KUKA KRL program: MyProgram_304().src

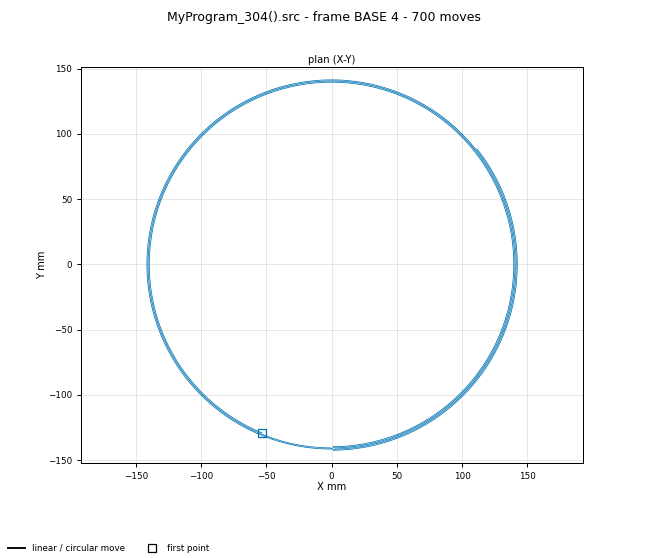
[picture p0: tool path of MyProgram_304().src in frame BASE 4, 700 of 700 moves have a stored position in this frame; points joined in program order, loops and branches not executed]
&ACCESS RVP
&REL 1
&PARAM TEMPLATE = C:\KRC\Roboter\Template\vorgabe
&PARAM EDITMASK = *
DEF MyProgram_304()
; ---- Setting reference (Base) ----
$BASE = BASE_DATA[4]

; --------------------------
; ---- Setting tool (TCP) ----
$TOOL = TOOL_DATA[3]
; --------------------------

$VEL.CP = VEL_APROX_PRINT
Startdeposition()
$VEL.CP = VEL_PRINT
LIN {X -53.4181,Y -129.0788,Z 180,A -108.7523,B 5.3109,C 0.3866,E1 5.2646,E2 201.3046} C_DIS
LIN {X -56.4505,Y -127.7825,Z 180,A -110.2013,B 5.3109,C 0.3863,E1 5.2608,E2 202.7664} C_DIS
LIN {X -60.7814,Y -125.7801,Z 180,A -112.5486,B 5.3109,C 0.3883,E1 5.2548,E2 205.165} C_DIS
LIN {X -64.8227,Y -123.7443,Z 180,A -113.8658,B 5.3114,C 0.3803,E1 5.2517,E2 206.4117} C_DIS
LIN {X -68.8662,Y -121.5434,Z 180,A -115.942,B 5.3114,C 0.3799,E1 5.2465,E2 208.5128} C_DIS
LIN {X -72.8889,Y -119.1739,Z 180,A -117.7837,B 5.3117,C 0.3765,E1 5.2422,E2 210.3448} C_DIS
LIN {X -75.6245,Y -117.4571,Z 180,A -119.198,B 5.3117,C 0.3756,E1 5.2388,E2 211.7709} C_DIS
LIN {X -78.8968,Y -115.2844,Z 180,A -121.1686,B 5.3117,C 0.3769,E1 5.2341,E2 213.7885} C_DIS
LIN {X -82.2269,Y -112.9324,Z 180,A -122.773,B 5.3119,C 0.3735,E1 5.2305,E2 215.384} C_DIS
LIN {X -85.2034,Y -110.7056,Z 180,A -124.0807,B 5.3122,C 0.3688,E1 5.2277,E2 216.6631} C_DIS
LIN {X -88.7338,Y -107.8966,Z 180,A -125.9867,B 5.3124,C 0.3662,E1 5.2235,E2 218.5762} C_DIS
LIN {X -92.192,Y -104.9572,Z 180,A -127.8448,B 5.3126,C 0.3629,E1 5.2196,E2 220.4335} C_DIS
LIN {X -95.4577,Y -101.9958,Z 180,A -129.699,B 5.3128,C 0.36,E1 5.2158,E2 222.2935} C_DIS
LIN {X -98.7586,Y -98.8033,Z 180,A -131.5928,B 5.313,C 0.3565,E1 5.212,E2 224.1882} C_DIS
LIN {X -101.9125,Y -95.5469,Z 180,A -133.5295,B 5.3132,C 0.3536,E1 5.2083,E2 226.1346} C_DIS
LIN {X -105.0138,Y -92.1271,Z 180,A -135.4558,B 5.3135,C 0.35,E1 5.2047,E2 228.0647} C_DIS
LIN {X -107.866,Y -88.7709,Z 180,A -137.2983,B 5.3137,C 0.3465,E1 5.2014,E2 229.9114} C_DIS
LIN {X -110.7145,Y -85.1918,Z 180,A -138.9304,B 5.3141,C 0.3401,E1 5.1986,E2 231.5111} C_DIS
LIN {X -112.3282,Y -83.0519,Z 180,A -140.3289,B 5.3141,C 0.3405,E1 5.1962,E2 232.9482} C_DIS
LIN {X -114.9154,Y -79.4344,Z 180,A -142.1992,B 5.3143,C 0.3368,E1 5.1932,E2 234.8238} C_DIS
LIN {X -116.9571,Y -76.3961,Z 180,A -143.832,B 5.3145,C 0.3345,E1 5.1907,E2 236.4731} C_DIS
LIN {X -119.7431,Y -71.9508,Z 180,A -145.7127,B 5.3149,C 0.3269,E1 5.188,E2 238.3177} C_DIS
LIN {X -122.8692,Y -66.4714,Z 180,A -148.6944,B 5.3151,C 0.3242,E1 5.1838,E2 241.3494} C_DIS
LIN {X -125.0963,Y -62.1747,Z 180,A -150.5037,B 5.3155,C 0.3177,E1 5.1816,E2 243.1351} C_DIS
LIN {X -126.6631,Y -58.9167,Z 180,A -152.1928,B 5.3156,C 0.3158,E1 5.1795,E2 244.8501} C_DIS
LIN {X -128.6518,Y -54.4406,Z 180,A -154.1647,B 5.3159,C 0.3103,E1 5.1773,E2 246.8163} C_DIS
LIN {X -129.8644,Y -51.4832,Z 180,A -155.7497,B 5.3159,C 0.3093,E1 5.1757,E2 248.4359} C_DIS
LIN {X -131.0841,Y -48.2916,Z 180,A -157.1548,B 5.3162,C 0.3056,E1 5.1743,E2 249.8406} C_DIS
LIN {X -132.1648,Y -45.2484,Z 180,A -158.3647,B 5.3165,C 0.3011,E1 5.1732,E2 251.035} C_DIS
LIN {X -133.3531,Y -41.62,Z 180,A -159.865,B 5.3167,C 0.2963,E1 5.1719,E2 252.5261} C_DIS
LIN {X -134.4327,Y -37.9823,Z 180,A -161.4301,B 5.317,C 0.2921,E1 5.1707,E2 254.0912} C_DIS
LIN {X -135.3964,Y -34.3875,Z 180,A -163.0135,B 5.3172,C 0.2885,E1 5.1696,E2 255.681} C_DIS
LIN {X -136.1324,Y -31.3482,Z 180,A -164.2721,B 5.3174,C 0.2847,E1 5.1688,E2 256.9357} C_DIS
LIN {X -136.8639,Y -27.9821,Z 180,A -165.5232,B 5.3176,C 0.2794,E1 5.1681,E2 258.1651} C_DIS
LIN {X -137.4255,Y -25.0834,Z 180,A -166.9887,B 5.3177,C 0.2783,E1 5.1673,E2 259.6626} C_DIS
LIN {X -138.0139,Y -21.6086,Z 180,A -168.4852,B 5.3179,C 0.2747,E1 5.1666,E2 261.1647} C_DIS
LIN {X -138.4562,Y -18.5685,Z 180,A -169.9672,B 5.3179,C 0.2731,E1 5.166,E2 262.6742} C_DIS
LIN {X -139.2639,Y -10.996,Z 180,A -173.1053,B 5.3184,C 0.2644,E1 5.1652,E2 265.812} C_DIS
LIN {X -139.4901,Y -7.5904,Z 180,A -174.8697,B 5.3184,C 0.2636,E1 5.1649,E2 267.6217} C_DIS
LIN {X -139.6482,Y -3.635,Z 180,A -175.7772,B 5.319,C 0.2527,E1 5.1649,E2 268.4367} C_DIS
LIN {X -139.6884,Y 1.5471,Z 180,A -178.478,B 5.319,C 0.2517,E1 5.1649,E2 271.2095} C_DIS
LIN {X -139.3259,Y 10.151,Z 180,A 178.1814,B 5.3196,C 0.24,E1 5.1653,E2 274.523} C_DIS
LIN {X -138.7226,Y 16.4559,Z 180,A 175.3926,B 5.3198,C 0.2343,E1 5.166,E2 277.3342} C_DIS
LIN {X -138.2382,Y 20.1258,Z 180,A 173.8815,B 5.32,C 0.2299,E1 5.1666,E2 278.8431} C_DIS
LIN {X -137.7937,Y 22.9699,Z 180,A 172.4203,B 5.32,C 0.229,E1 5.1673,E2 280.3389} C_DIS
LIN {X -136.6551,Y 28.9886,Z 180,A 170.1284,B 5.3204,C 0.2201,E1 5.1685,E2 282.6008} C_DIS
LIN {X -135.9071,Y 32.3133,Z 180,A 168.5489,B 5.3205,C 0.2178,E1 5.1695,E2 284.2022} C_DIS
LIN {X -135.0439,Y 35.7475,Z 180,A 167.0737,B 5.3207,C 0.214,E1 5.1705,E2 285.679} C_DIS
LIN {X -134.221,Y 38.7258,Z 180,A 165.7742,B 5.3207,C 0.2108,E1 5.1715,E2 286.9816} C_DIS
LIN {X -133.127,Y 42.3307,Z 180,A 164.1851,B 5.3209,C 0.207,E1 5.1729,E2 288.5749} C_DIS
LIN {X -131.7274,Y 46.5099,Z 180,A 162.2401,B 5.3211,C 0.2033,E1 5.1746,E2 290.5357} C_DIS
LIN {X -130.6009,Y 49.5825,Z 180,A 160.8237,B 5.3211,C 0.2004,E1 5.1761,E2 291.9603} C_DIS
LIN {X -128.5842,Y 54.6025,Z 180,A 158.5967,B 5.3214,C 0.1946,E1 5.1784,E2 294.1864} C_DIS
LIN {X -126.939,Y 58.3201,Z 180,A 157.2078,B 5.3217,C 0.1878,E1 5.18,E2 295.5387} C_DIS
LIN {X -125.701,Y 60.9469,Z 180,A 155.4772,B 5.3216,C 0.1895,E1 5.1821,E2 297.3362} C_DIS
LIN {X -124.2165,Y 63.9159,Z 180,A 154.1121,B 5.3217,C 0.1861,E1 5.1839,E2 298.7005} C_DIS
LIN {X -122.6686,Y 66.8402,Z 180,A 152.908,B 5.3219,C 0.1814,E1 5.1854,E2 299.8843} C_DIS
LIN {X -120.3453,Y 70.9383,Z 180,A 150.9383,B 5.322,C 0.1769,E1 5.1882,E2 301.8571} C_DIS
LIN {X -117.9862,Y 74.7965,Z 180,A 149.0261,B 5.3222,C 0.173,E1 5.191,E2 303.7748} C_DIS
LIN {X -115.4538,Y 78.6496,Z 180,A 147.077,B 5.3222,C 0.169,E1 5.1941,E2 305.7295} C_DIS
LIN {X -112.8106,Y 82.3959,Z 180,A 145.3761,B 5.3225,C 0.163,E1 5.1968,E2 307.4063} C_DIS
LIN {X -110.0024,Y 86.1086,Z 180,A 143.1989,B 5.3225,C 0.1612,E1 5.2005,E2 309.6154} C_DIS
LIN {X -107.1393,Y 89.6459,Z 180,A 141.4016,B 5.3227,C 0.1565,E1 5.2037,E2 311.4025} C_DIS
LIN {X -103.7343,Y 93.5651,Z 180,A 138.6523,B 5.3227,C 0.1577,E1 5.209,E2 314.227} C_DIS
LIN {X -100.4211,Y 97.1123,Z 180,A 137.1074,B 5.3229,C 0.1495,E1 5.2118,E2 315.715} C_DIS
LIN {X -97.8974,Y 99.6558,Z 180,A 135.0674,B 5.3228,C 0.1519,E1 5.216,E2 317.8245} C_DIS
LIN {X -94.1292,Y 103.223,Z 180,A 132.9812,B 5.3229,C 0.1475,E1 5.2203,E2 319.9038} C_DIS
LIN {X -90.597,Y 106.3362,Z 180,A 131.4762,B 5.3231,C 0.1399,E1 5.2234,E2 321.3544} C_DIS
LIN {X -87.0706,Y 109.2423,Z 180,A 129.612,B 5.3232,C 0.1364,E1 5.2274,E2 323.2158} C_DIS
LIN {X -84.1015,Y 111.5443,Z 180,A 127.5305,B 5.3232,C 0.1391,E1 5.2322,E2 325.3631} C_DIS
LIN {X -80.1977,Y 114.3838,Z 180,A 125.9877,B 5.3233,C 0.1316,E1 5.2356,E2 326.8502} C_DIS
LIN {X -76.4605,Y 116.9152,Z 180,A 124.1034,B 5.3234,C 0.129,E1 5.24,E2 328.7372} C_DIS
LIN {X -72.6594,Y 119.3147,Z 180,A 122.36,B 5.3234,C 0.1253,E1 5.2441,E2 330.4667} C_DIS
LIN {X -69.4823,Y 121.1919,Z 180,A 120.6836,B 5.3235,C 0.1248,E1 5.2482,E2 332.1622} C_DIS
LIN {X -65.5195,Y 123.3784,Z 180,A 118.8849,B 5.3235,C 0.1218,E1 5.2526,E2 333.9523} C_DIS
LIN {X -62.1192,Y 125.1237,Z 180,A 117.2852,B 5.3236,C 0.1201,E1 5.2566,E2 335.5548} C_DIS
LIN {X -57.8735,Y 127.1455,Z 180,A 115.2756,B 5.3236,C 0.1187,E1 5.2617,E2 337.5732} C_DIS
LIN {X -51.9459,Y 129.6779,Z 180,A 112.3818,B 5.3236,C 0.1185,E1 5.2692,E2 340.496} C_DIS
LIN {X -48.6279,Y 130.9585,Z 180,A 111.18,B 5.3237,C 0.1144,E1 5.2723,E2 341.665} C_DIS
LIN {X -44.4366,Y 132.4392,Z 180,A 109.372,B 5.3237,C 0.1126,E1 5.277,E2 343.4699} C_DIS
LIN {X -41.3217,Y 133.4443,Z 180,A 108.0284,B 5.3237,C 0.1115,E1 5.2806,E2 344.8128} C_DIS
LIN {X -38.2459,Y 134.359,Z 180,A 106.3124,B 5.3237,C 0.1148,E1 5.2854,E2 346.5775} C_DIS
LIN {X -34.5071,Y 135.366,Z 180,A 105.1143,B 5.3238,C 0.1096,E1 5.2885,E2 347.7263} C_DIS
LIN {X -31.3524,Y 136.1315,Z 180,A 103.7636,B 5.3238,C 0.109,E1 5.2921,E2 349.0787} C_DIS
LIN {X -28.0893,Y 136.8421,Z 180,A 102.2931,B 5.3238,C 0.1093,E1 5.2962,E2 350.5609} C_DIS
LIN {X -19.2145,Y 138.3685,Z 180,A 98.5818,B 5.3238,C 0.108,E1 5.3064,E2 354.2724} C_DIS
LIN {X -15.0864,Y 138.8782,Z 180,A 96.9214,B 5.3238,C 0.107,E1 5.311,E2 355.9262} C_DIS
LIN {X -9.6565,Y 139.362,Z 180,A 94.5696,B 5.3238,C 0.1079,E1 5.3176,E2 358.2914} C_DIS
LIN {X -5.0259,Y 139.6055,Z 180,A 92.8427,B 5.3239,C 0.1057,E1 5.3224,E2 359.9957} C_DIS
LIN {X -1.2399,Y 139.6906,Z 180,A 91.2064,B 5.3239,C 0.1067,E1 5.327,E2 361.6416} C_DIS
LIN {X 3.0957,Y 139.6631,Z 180,A 89.4454,B 5.3239,C 0.1067,E1 5.3319,E2 363.3998} C_DIS
LIN {X 6.8555,Y 139.527,Z 180,A 87.9816,B 5.3239,C 0.1059,E1 5.3359,E2 364.853} C_DIS
LIN {X 10.1316,Y 139.3273,Z 180,A 86.6321,B 5.3239,C 0.1063,E1 5.3397,E2 366.2023} C_DIS
LIN {X 13.9379,Y 138.9994,Z 180,A 84.9893,B 5.3239,C 0.1077,E1 5.3443,E2 367.854} C_DIS
LIN {X 17.3009,Y 138.6217,Z 180,A 83.4925,B 5.3239,C 0.1095,E1 5.3485,E2 369.3639} C_DIS
LIN {X 23.4985,Y 137.7055,Z 180,A 81.0194,B 5.3239,C 0.1095,E1 5.3553,E2 371.8242} C_DIS
LIN {X 27.313,Y 137,Z 180,A 79.39,B 5.3239,C 0.111,E1 5.3597,E2 373.4579} C_DIS
LIN {X 31.8403,Y 136.0189,Z 180,A 77.378,B 5.3238,C 0.1136,E1 5.3653,E2 375.4832} C_DIS
LIN {X 35.117,Y 135.2112,Z 180,A 76.2143,B 5.3238,C 0.1119,E1 5.3683,E2 376.6193} C_DIS
LIN {X 38.9715,Y 134.1491,Z 180,A 74.6646,B 5.3238,C 0.1121,E1 5.3725,E2 378.1573} C_DIS
LIN {X 41.8856,Y 133.2692,Z 180,A 73.3079,B 5.3238,C 0.1146,E1 5.3761,E2 379.5274} C_DIS
LIN {X 46.6217,Y 131.6879,Z 180,A 71.2783,B 5.3237,C 0.1163,E1 5.3815,E2 381.5543} C_DIS
LIN {X 50.0811,Y 130.4103,Z 180,A 69.8417,B 5.3237,C 0.1169,E1 5.3852,E2 382.9812} C_DIS
LIN {X 53.5107,Y 129.0401,Z 180,A 68.3385,B 5.3237,C 0.1185,E1 5.3891,E2 384.4828} C_DIS
LIN {X 56.8677,Y 127.5959,Z 180,A 67.0037,B 5.3237,C 0.1181,E1 5.3924,E2 385.7969} C_DIS
LIN {X 62.2697,Y 125.0495,Z 180,A 64.5146,B 5.3236,C 0.1217,E1 5.3987,E2 388.2908} C_DIS
LIN {X 66.0051,Y 123.12,Z 180,A 62.6956,B 5.3235,C 0.1253,E1 5.4033,E2 390.1216} C_DIS
LIN {X 70.0877,Y 120.8425,Z 180,A 60.8254,B 5.3235,C 0.1274,E1 5.4078,E2 391.9859} C_DIS
LIN {X 74.0028,Y 118.4856,Z 180,A 58.9975,B 5.3234,C 0.1296,E1 5.4121,E2 393.808} C_DIS
LIN {X 77.581,Y 116.1739,Z 180,A 56.9544,B 5.3232,C 0.1364,E1 5.417,E2 395.8882} C_DIS
LIN {X 80.7286,Y 114.0094,Z 180,A 55.6359,B 5.3232,C 0.1356,E1 5.4199,E2 397.1758} C_DIS
LIN {X 84.5976,Y 111.169,Z 180,A 53.724,B 5.3232,C 0.1382,E1 5.4242,E2 399.0807} C_DIS
LIN {X 88.2382,Y 108.3016,Z 180,A 51.827,B 5.3231,C 0.1416,E1 5.4283,E2 400.9775} C_DIS
LIN {X 92.0568,Y 105.0752,Z 180,A 49.9356,B 5.3231,C 0.1433,E1 5.4323,E2 402.8493} C_DIS
LIN {X 94.5696,Y 102.8191,Z 180,A 47.9785,B 5.3227,C 0.1539,E1 5.4365,E2 404.8782} C_DIS
LIN {X 98.3552,Y 99.2041,Z 180,A 46.3995,B 5.3228,C 0.1503,E1 5.4395,E2 406.3866} C_DIS
LIN {X 101.5988,Y 95.8794,Z 180,A 44.5516,B 5.3228,C 0.1534,E1 5.443,E2 408.2278} C_DIS
LIN {X 104.6892,Y 92.4951,Z 180,A 42.7152,B 5.3227,C 0.1568,E1 5.4465,E2 410.0592} C_DIS
LIN {X 107.1038,Y 89.6882,Z 180,A 40.9069,B 5.3224,C 0.1642,E1 5.4498,E2 411.9043} C_DIS
LIN {X 109.6071,Y 86.6119,Z 180,A 39.586,B 5.3224,C 0.1635,E1 5.452,E2 413.1873} C_DIS
LIN {X 112.3135,Y 83.0726,Z 180,A 37.8081,B 5.3224,C 0.167,E1 5.455,E2 414.9596} C_DIS
LIN {X 114.8587,Y 79.5158,Z 180,A 36.1736,B 5.3223,C 0.1689,E1 5.4576,E2 416.5745} C_DIS
LIN {X 116.9308,Y 76.4366,Z 180,A 34.5411,B 5.3221,C 0.1741,E1 5.4601,E2 418.2216} C_DIS
LIN {X 118.9321,Y 73.2831,Z 180,A 32.8039,B 5.3219,C 0.1808,E1 5.4627,E2 419.9854} C_DIS
LIN {X 120.8792,Y 70.0239,Z 180,A 31.4886,B 5.3219,C 0.1811,E1 5.4645,E2 421.2707} C_DIS
LIN {X 123.2434,Y 65.7753,Z 180,A 29.5782,B 5.3218,C 0.1849,E1 5.4671,E2 423.1714} C_DIS
LIN {X 125.0282,Y 62.3128,Z 180,A 28.2508,B 5.3218,C 0.1849,E1 5.4687,E2 424.4651} C_DIS
LIN {X 126.6486,Y 58.948,Z 180,A 26.6413,B 5.3216,C 0.1901,E1 5.4706,E2 426.0853} C_DIS
LIN {X 128.0692,Y 55.7949,Z 180,A 25.4362,B 5.3216,C 0.1906,E1 5.472,E2 427.2639} C_DIS
LIN {X 130.2404,Y 50.5183,Z 180,A 23.0133,B 5.3213,C 0.198,E1 5.4746,E2 429.6986} C_DIS
LIN {X 131.3973,Y 47.4278,Z 180,A 21.7673,B 5.3213,C 0.2,E1 5.4757,E2 430.9317} C_DIS
LIN {X 132.4219,Y 44.4886,Z 180,A 20.423,B 5.321,C 0.2045,E1 5.477,E2 432.2854} C_DIS
LIN {X 133.5287,Y 41.046,Z 180,A 18.9479,B 5.3209,C 0.2084,E1 5.4782,E2 433.7603} C_DIS
LIN {X 134.5026,Y 37.7326,Z 180,A 17.6107,B 5.3208,C 0.2111,E1 5.4792,E2 435.0882} C_DIS
LIN {X 135.3467,Y 34.5835,Z 180,A 16.2761,B 5.3206,C 0.2147,E1 5.4802,E2 436.4233} C_DIS
LIN {X 136.0439,Y 31.7359,Z 180,A 15.1574,B 5.3206,C 0.2168,E1 5.4809,E2 437.532} C_DIS
LIN {X 136.9679,Y 27.471,Z 180,A 13.2708,B 5.3203,C 0.2232,E1 5.482,E2 439.4322} C_DIS
LIN {X 137.6674,Y 23.727,Z 180,A 11.1723,B 5.3198,C 0.2356,E1 5.483,E2 441.6003} C_DIS
LIN {X 138.492,Y 18.2952,Z 180,A 9.5426,B 5.3198,C 0.2326,E1 5.4836,E2 443.1519} C_DIS
LIN {X 139.0361,Y 13.5554,Z 180,A 7.728,B 5.3198,C 0.236,E1 5.4841,E2 444.9496} C_DIS
LIN {X 139.3314,Y 10.0758,Z 180,A 6.3138,B 5.3196,C 0.2398,E1 5.4844,E2 446.3625} C_DIS
LIN {X 139.5729,Y 5.8598,Z 180,A 4.6384,B 5.3194,C 0.2439,E1 5.4847,E2 448.0319} C_DIS
LIN {X 139.6755,Y 2.3565,Z 180,A 3.267,B 5.3192,C 0.247,E1 5.4847,E2 449.3957} C_DIS
LIN {X 139.6814,Y -1.9962,Z 180,A 1.495,B 5.319,C 0.2519,E1 5.4847,E2 451.1675} C_DIS
LIN {X 139.5624,Y -6.1305,Z 180,A -0.2183,B 5.3188,C 0.257,E1 5.4846,E2 452.8842} C_DIS
LIN {X 139.3144,Y -10.3093,Z 180,A -1.8235,B 5.3186,C 0.2602,E1 5.4843,E2 454.4764} C_DIS
LIN {X 138.932,Y -14.5868,Z 180,A -3.5823,B 5.3184,C 0.2651,E1 5.4838,E2 456.2362} C_DIS
LIN {X 138.4803,Y -18.3843,Z 180,A -5.0577,B 5.3182,C 0.2682,E1 5.4833,E2 457.7008} C_DIS
LIN {X 137.8848,Y -22.4237,Z 180,A -7.1758,B 5.3176,C 0.2796,E1 5.4823,E2 459.8776} C_DIS
LIN {X 137.0513,Y -27.0612,Z 180,A -8.6435,B 5.3177,C 0.278,E1 5.4816,E2 461.287} C_DIS
LIN {X 136.2801,Y -30.7018,Z 180,A -10.0627,B 5.3176,C 0.2807,E1 5.4807,E2 462.6935} C_DIS
LIN {X 134.9928,Y -35.9392,Z 180,A -12.0724,B 5.3174,C 0.2837,E1 5.4794,E2 464.6787} C_DIS
LIN {X 133.1515,Y -42.2542,Z 180,A -14.8183,B 5.317,C 0.2919,E1 5.4772,E2 467.4332} C_DIS
LIN {X 132.0483,Y -45.5842,Z 180,A -16.2158,B 5.3168,C 0.2952,E1 5.476,E2 468.8266} C_DIS
LIN {X 130.9944,Y -48.5319,Z 180,A -17.5271,B 5.3166,C 0.2991,E1 5.4747,E2 470.1426} C_DIS
LIN {X 129.6758,Y -51.951,Z 180,A -18.8882,B 5.3165,C 0.301,E1 5.4733,E2 471.4864} C_DIS
LIN {X 128.3506,Y -55.144,Z 180,A -20.2885,B 5.3163,C 0.3045,E1 5.4718,E2 472.8857} C_DIS
LIN {X 126.9225,Y -58.3557,Z 180,A -21.7176,B 5.3161,C 0.3081,E1 5.4702,E2 474.3145} C_DIS
LIN {X 125.5516,Y -61.2518,Z 180,A -23.069,B 5.3158,C 0.312,E1 5.4685,E2 475.6719} C_DIS
LIN {X 123.7294,Y -64.8509,Z 180,A -24.6078,B 5.3157,C 0.3146,E1 5.4666,E2 477.197} C_DIS
LIN {X 121.6076,Y -68.7525,Z 180,A -26.4799,B 5.3154,C 0.3199,E1 5.464,E2 479.0774} C_DIS
LIN {X 119.4654,Y -72.4101,Z 180,A -28.5865,B 5.3148,C 0.3297,E1 5.4609,E2 481.2336} C_DIS
LIN {X 117.0766,Y -76.212,Z 180,A -29.9613,B 5.3149,C 0.3273,E1 5.459,E2 482.5491} C_DIS
LIN {X 114.5875,Y -79.9056,Z 180,A -31.6688,B 5.3148,C 0.3299,E1 5.4563,E2 484.2426} C_DIS
LIN {X 112.2867,Y -83.1086,Z 180,A -33.9984,B 5.3139,C 0.3442,E1 5.4523,E2 486.6666} C_DIS
LIN {X 108.717,Y -87.7256,Z 180,A -35.6708,B 5.3142,C 0.3391,E1 5.4495,E2 488.2471} C_DIS
LIN {X 105.9713,Y -91.0236,Z 180,A -37.3819,B 5.314,C 0.3423,E1 5.4464,E2 489.9533} C_DIS
LIN {X 104.0082,Y -93.2603,Z 180,A -38.6493,B 5.3138,C 0.3457,E1 5.4441,E2 491.2279} C_DIS
LIN {X 101.3904,Y -96.1003,Z 180,A -40.1605,B 5.3136,C 0.348,E1 5.4412,E2 492.7309} C_DIS
LIN {X 98.3275,Y -99.2317,Z 180,A -41.8803,B 5.3134,C 0.3507,E1 5.4378,E2 494.4421} C_DIS
LIN {X 95.3265,Y -102.1179,Z 180,A -43.6035,B 5.3132,C 0.3544,E1 5.4343,E2 496.1689} C_DIS
LIN {X 92.019,Y -105.1082,Z 180,A -45.2382,B 5.3132,C 0.3552,E1 5.431,E2 497.7796} C_DIS
LIN {X 89.2239,Y -107.4909,Z 180,A -46.8661,B 5.3128,C 0.3598,E1 5.4275,E2 499.4248} C_DIS
LIN {X 85.8046,Y -110.2399,Z 180,A -48.3533,B 5.3128,C 0.3587,E1 5.4243,E2 500.8722} C_DIS
LIN {X 83.6515,Y -111.8824,Z 180,A -49.6148,B 5.3126,C 0.3629,E1 5.4214,E2 502.1547} C_DIS
LIN {X 79.6876,Y -114.7392,Z 180,A -51.7708,B 5.3122,C 0.3685,E1 5.4165,E2 504.3323} C_DIS
LIN {X 75.6663,Y -117.4307,Z 180,A -53.9476,B 5.3118,C 0.3745,E1 5.4113,E2 506.536} C_DIS
LIN {X 72.4638,Y -119.4329,Z 180,A -54.965,B 5.3122,C 0.3695,E1 5.4091,E2 507.4846} C_DIS
LIN {X 67.1571,Y -122.4957,Z 180,A -57.6945,B 5.3117,C 0.3763,E1 5.4024,E2 510.2447} C_DIS
LIN {X 63.5525,Y -124.4015,Z 180,A -59.2118,B 5.3117,C 0.3765,E1 5.3987,E2 511.7428} C_DIS
LIN {X 60.3887,Y -125.9677,Z 180,A -60.674,B 5.3115,C 0.3787,E1 5.395,E2 513.208} C_DIS
LIN {X 57.1271,Y -127.4799,Z 180,A -61.9984,B 5.3115,C 0.3786,E1 5.3917,E2 514.5136} C_DIS
LIN {X 54.1683,Y -128.7655,Z 180,A -63.3875,B 5.3113,C 0.3811,E1 5.3881,E2 515.9124} C_DIS
LIN {X 50.9744,Y -130.063,Z 180,A -64.8485,B 5.3112,C 0.3834,E1 5.3843,E2 517.3806} C_DIS
LIN {X 47.7036,Y -131.2979,Z 180,A -66.2567,B 5.3111,C 0.3846,E1 5.3806,E2 518.7865} C_DIS
LIN {X 44.2513,Y -132.5009,Z 180,A -67.7178,B 5.3111,C 0.3856,E1 5.3767,E2 520.2435} C_DIS
LIN {X 41.1267,Y -133.504,Z 180,A -68.8889,B 5.3111,C 0.3846,E1 5.3737,E2 521.3923} C_DIS
LIN {X 37.023,Y -134.701,Z 180,A -70.8902,B 5.3107,C 0.3895,E1 5.3682,E2 523.4278} C_DIS
LIN {X 30.5957,Y -136.3043,Z 180,A -73.5088,B 5.3107,C 0.3904,E1 5.3611,E2 526.0351} C_DIS
LIN {X 23.7366,Y -137.6657,Z 180,A -76.8393,B 5.3101,C 0.3982,E1 5.3518,E2 529.4284} C_DIS
LIN {X 19.4208,Y -138.339,Z 180,A -78.1847,B 5.3104,C 0.3934,E1 5.3483,E2 530.7159} C_DIS
LIN {X 15.4627,Y -138.8377,Z 180,A -79.8042,B 5.3104,C 0.394,E1 5.3438,E2 532.3341} C_DIS
LIN {X 11.8735,Y -139.1897,Z 180,A -81.2565,B 5.3104,C 0.3942,E1 5.3397,E2 533.7836} C_DIS
LIN {X 7.819,Y -139.4783,Z 180,A -82.9889,B 5.3103,C 0.3955,E1 5.3349,E2 535.5256} C_DIS
LIN {X 3.6418,Y -139.648,Z 180,A -84.6179,B 5.3103,C 0.3949,E1 5.3304,E2 537.1441} C_DIS
LIN {X 0.988,Y -139.6903,Z 180,A -85.5323,B 5.3105,C 0.3929,E1 5.3279,E2 538.0358} C_DIS
Enddeposition()
LIN {X 0.988,Y -139.6903,Z 180,A -85.5323,B 5.3105,C 0.3929,E1 5.3279,E2 538.0358} C_DIS
Startdeposition()
$VEL.CP = VEL_PRINT
LIN {X 1.6591,Y -140.5898,Z 180,A -84.529,B 5.0673,C 0.3825,E1 5.0873,E2 537.0364} C_DIS
LIN {X 5.6051,Y -140.4862,Z 180,A -83.0223,B 5.0673,C 0.3834,E1 5.0914,E2 535.5427} C_DIS
LIN {X 9.7167,Y -140.2627,Z 180,A -81.2945,B 5.0673,C 0.3822,E1 5.0963,E2 533.8074} C_DIS
LIN {X 13.6344,Y -139.9353,Z 180,A -79.7585,B 5.0673,C 0.3824,E1 5.1005,E2 532.2794} C_DIS
LIN {X 17.757,Y -139.4729,Z 180,A -77.6117,B 5.0678,C 0.3759,E1 5.1067,E2 530.0698} C_DIS
LIN {X 22.0608,Y -138.8573,Z 180,A -76.277,B 5.0675,C 0.3804,E1 5.1102,E2 528.7934} C_DIS
LIN {X 26.0361,Y -138.1665,Z 180,A -74.5889,B 5.0675,C 0.3788,E1 5.1148,E2 527.0984} C_DIS
LIN {X 29.9679,Y -137.3671,Z 180,A -72.4377,B 5.0682,C 0.3711,E1 5.1209,E2 524.876} C_DIS
LIN {X 35.0666,Y -136.1553,Z 180,A -70.9688,B 5.0677,C 0.3779,E1 5.1247,E2 523.4964} C_DIS
LIN {X 38.4418,Y -135.2415,Z 180,A -69.2728,B 5.068,C 0.3732,E1 5.1293,E2 521.7628} C_DIS
LIN {X 43.0773,Y -133.8361,Z 180,A -67.5594,B 5.0679,C 0.3746,E1 5.1338,E2 520.0833} C_DIS
LIN {X 46.4412,Y -132.7066,Z 180,A -66.135,B 5.0679,C 0.3734,E1 5.1375,E2 518.6608} C_DIS
LIN {X 49.962,Y -131.4227,Z 180,A -64.6541,B 5.0681,C 0.3723,E1 5.1414,E2 517.1851} C_DIS
LIN {X 52.7883,Y -130.3115,Z 180,A -63.3956,B 5.0681,C 0.3706,E1 5.1447,E2 515.9228} C_DIS
LIN {X 56.5308,Y -128.7344,Z 180,A -61.7768,B 5.0683,C 0.369,E1 5.1488,E2 514.3078} C_DIS
LIN {X 59.2753,Y -127.4918,Z 180,A -60.5485,B 5.0684,C 0.3674,E1 5.1519,E2 513.0785} C_DIS
LIN {X 62.7104,Y -125.8386,Z 180,A -59.0283,B 5.0685,C 0.3658,E1 5.1558,E2 511.5616} C_DIS
LIN {X 65.3966,Y -124.4624,Z 180,A -57.847,B 5.0686,C 0.3647,E1 5.1587,E2 510.3859} C_DIS
LIN {X 69.9432,Y -121.9681,Z 180,A -55.4729,B 5.0691,C 0.358,E1 5.1645,E2 507.975} C_DIS
LIN {X 75.4813,Y -118.6209,Z 180,A -53.3038,B 5.0689,C 0.3602,E1 5.1696,E2 505.867} C_DIS
LIN {X 78.1143,Y -116.9032,Z 180,A -51.3428,B 5.0697,C 0.3487,E1 5.1743,E2 503.813} C_DIS
LIN {X 82.015,Y -114.2005,Z 180,A -49.8294,B 5.0696,C 0.3512,E1 5.1777,E2 502.3551} C_DIS
LIN {X 85.9243,Y -111.2891,Z 180,A -47.9606,B 5.0697,C 0.3492,E1 5.1818,E2 500.5005} C_DIS
LIN {X 89.0765,Y -108.7823,Z 180,A -46.359,B 5.0699,C 0.3467,E1 5.1852,E2 498.9029} C_DIS
LIN {X 92.8247,Y -105.6026,Z 180,A -44.3228,B 5.0702,C 0.3424,E1 5.1896,E2 496.8605} C_DIS
LIN {X 96.2359,Y -102.5035,Z 180,A -42.5076,B 5.0704,C 0.3395,E1 5.1933,E2 495.0522} C_DIS
LIN {X 99.4726,Y -99.3657,Z 180,A -40.6808,B 5.0706,C 0.3358,E1 5.1969,E2 493.2252} C_DIS
LIN {X 103.7158,Y -94.9276,Z 180,A -38.2282,B 5.0709,C 0.3312,E1 5.2016,E2 490.7772} C_DIS
LIN {X 106.7536,Y -91.4985,Z 180,A -36.4138,B 5.0711,C 0.3278,E1 5.2049,E2 488.9681} C_DIS
LIN {X 109.6839,Y -87.9646,Z 180,A -34.3051,B 5.0716,C 0.3201,E1 5.2087,E2 486.8258} C_DIS
LIN {X 112.0988,Y -84.8651,Z 180,A -32.9868,B 5.0716,C 0.3205,E1 5.2108,E2 485.5441} C_DIS
LIN {X 117.0782,Y -77.8522,Z 180,A -29.8517,B 5.0718,C 0.3175,E1 5.2158,E2 482.4557} C_DIS
LIN {X 120.6294,Y -72.2276,Z 180,A -27.0992,B 5.0722,C 0.3103,E1 5.2199,E2 479.6954} C_DIS
LIN {X 122.5106,Y -68.9881,Z 180,A -25.4793,B 5.0725,C 0.3051,E1 5.2221,E2 478.0617} C_DIS
LIN {X 124.6716,Y -64.9983,Z 180,A -23.7439,B 5.0727,C 0.302,E1 5.2244,E2 476.3399} C_DIS
LIN {X 126.2382,Y -61.9003,Z 180,A -22.3939,B 5.0729,C 0.2993,E1 5.2261,E2 474.9972} C_DIS
LIN {X 127.7298,Y -58.7605,Z 180,A -20.9869,B 5.0731,C 0.2958,E1 5.2277,E2 473.5902} C_DIS
LIN {X 129.1559,Y -55.556,Z 180,A -19.5724,B 5.0733,C 0.2922,E1 5.2293,E2 472.1764} C_DIS
LIN {X 130.7266,Y -51.7586,Z 180,A -17.8413,B 5.0736,C 0.2869,E1 5.2311,E2 470.4364} C_DIS
LIN {X 132.1842,Y -47.9067,Z 180,A -16.3399,B 5.0737,C 0.285,E1 5.2326,E2 468.9571} C_DIS
LIN {X 133.353,Y -44.5496,Z 180,A -14.9465,B 5.0739,C 0.2819,E1 5.2338,E2 467.5698} C_DIS
LIN {X 134.8138,Y -39.9137,Z 180,A -12.6642,B 5.0744,C 0.272,E1 5.2357,E2 465.2457} C_DIS
LIN {X 135.8091,Y -36.3812,Z 180,A -10.9466,B 5.0748,C 0.2645,E1 5.2369,E2 463.4971} C_DIS
LIN {X 137.0637,Y -31.3248,Z 180,A -9.5821,B 5.0745,C 0.2699,E1 5.2378,E2 462.2319} C_DIS
LIN {X 138.6594,Y -23.2659,Z 180,A -6.4873,B 5.0748,C 0.2643,E1 5.2394,E2 459.1681} C_DIS
LIN {X 139.262,Y -19.3423,Z 180,A -4.6833,B 5.0752,C 0.257,E1 5.2401,E2 457.3383} C_DIS
LIN {X 139.7411,Y -15.5049,Z 180,A -3.0438,B 5.0755,C 0.2516,E1 5.2407,E2 455.6891} C_DIS
LIN {X 140.1172,Y -11.6184,Z 180,A -1.5954,B 5.0755,C 0.2492,E1 5.241,E2 454.2584} C_DIS
LIN {X 140.3475,Y -8.3912,Z 180,A -0.2573,B 5.0758,C 0.2451,E1 5.2413,E2 452.9167} C_DIS
LIN {X 140.5382,Y -4.1036,Z 180,A 1.4403,B 5.076,C 0.2409,E1 5.2415,E2 451.2244} C_DIS
LIN {X 140.6015,Y -0.0685,Z 180,A 3.1089,B 5.0762,C 0.2359,E1 5.2415,E2 449.5516} C_DIS
LIN {X 140.5487,Y 3.7249,Z 180,A 4.529,B 5.0763,C 0.2333,E1 5.2415,E2 448.1469} C_DIS
LIN {X 140.3989,Y 7.4915,Z 180,A 5.9684,B 5.0765,C 0.2304,E1 5.2412,E2 446.7191} C_DIS
LIN {X 140.1559,Y 11.1598,Z 180,A 7.5796,B 5.0767,C 0.2245,E1 5.2409,E2 445.0919} C_DIS
LIN {X 139.7915,Y 15.0361,Z 180,A 9.8258,B 5.0773,C 0.2102,E1 5.2402,E2 442.7573} C_DIS
LIN {X 138.9564,Y 21.4209,Z 180,A 11.3602,B 5.077,C 0.219,E1 5.2396,E2 441.365} C_DIS
LIN {X 138.4135,Y 24.6866,Z 180,A 12.8764,B 5.0772,C 0.2127,E1 5.2389,E2 439.8261} C_DIS
LIN {X 137.6453,Y 28.6688,Z 180,A 14.4278,B 5.0774,C 0.2096,E1 5.2381,E2 438.287} C_DIS
LIN {X 137.0158,Y 31.5344,Z 180,A 15.7867,B 5.0776,C 0.2039,E1 5.2372,E2 436.9059} C_DIS
LIN {X 135.71,Y 36.753,Z 180,A 17.7502,B 5.0777,C 0.2012,E1 5.2359,E2 434.971} C_DIS
LIN {X 134.8797,Y 39.6886,Z 180,A 19.0202,B 5.0779,C 0.1974,E1 5.2349,E2 433.6967} C_DIS
LIN {X 133.8341,Y 43.0836,Z 180,A 20.4031,B 5.0779,C 0.1944,E1 5.2337,E2 432.3215} C_DIS
LIN {X 132.5866,Y 46.7873,Z 180,A 21.946,B 5.0781,C 0.1909,E1 5.2323,E2 430.7843} C_DIS
LIN {X 130.1483,Y 53.1933,Z 180,A 24.6707,B 5.0783,C 0.1845,E1 5.2296,E2 428.067} C_DIS
LIN {X 128.9303,Y 56.0778,Z 180,A 25.9136,B 5.0784,C 0.1816,E1 5.2282,E2 426.8278} C_DIS
LIN {X 127.4724,Y 59.3172,Z 180,A 27.3389,B 5.0786,C 0.1782,E1 5.2265,E2 425.4047} C_DIS
LIN {X 125.9366,Y 62.5117,Z 180,A 28.7637,B 5.0786,C 0.1748,E1 5.2248,E2 423.9818} C_DIS
LIN {X 124.0201,Y 66.2369,Z 180,A 30.5188,B 5.0789,C 0.1698,E1 5.2225,E2 422.2197} C_DIS
LIN {X 120.7546,Y 72.0176,Z 180,A 32.7789,B 5.0789,C 0.1695,E1 5.2195,E2 420.0162} C_DIS
LIN {X 118.0141,Y 76.4257,Z 180,A 35.2036,B 5.0792,C 0.16,E1 5.2158,E2 417.5508} C_DIS
LIN {X 115.61,Y 80.0166,Z 180,A 36.8069,B 5.0792,C 0.1581,E1 5.2133,E2 415.9673} C_DIS
LIN {X 113.3688,Y 83.1608,Z 180,A 38.4344,B 5.0794,C 0.1537,E1 5.2106,E2 414.3322} C_DIS
LIN {X 110.7015,Y 86.6799,Z 180,A 40.3569,B 5.0795,C 0.1479,E1 5.2073,E2 412.3932} C_DIS
LIN {X 106.799,Y 91.4458,Z 180,A 42.6942,B 5.0796,C 0.1448,E1 5.2032,E2 410.0776} C_DIS
LIN {X 103.6067,Y 95.0466,Z 180,A 44.5014,B 5.0796,C 0.1427,E1 5.1998,E2 408.2898} C_DIS
LIN {X 100.7395,Y 98.0811,Z 180,A 46.283,B 5.0798,C 0.1381,E1 5.1964,E2 406.4975} C_DIS
LIN {X 96.1877,Y 102.5483,Z 180,A 49.0454,B 5.08,C 0.1307,E1 5.1907,E2 403.7135} C_DIS
LIN {X 93.4923,Y 105.0122,Z 180,A 50.0234,B 5.08,C 0.1348,E1 5.1889,E2 402.8009} C_DIS
LIN {X 90.1417,Y 107.9016,Z 180,A 51.9722,B 5.08,C 0.1294,E1 5.1847,E2 400.8331} C_DIS
LIN {X 86.8649,Y 110.5562,Z 180,A 53.711,B 5.0801,C 0.1261,E1 5.1809,E2 399.0915} C_DIS
LIN {X 83.2963,Y 113.2692,Z 180,A 55.7977,B 5.0803,C 0.1195,E1 5.1761,E2 396.9713} C_DIS
LIN {X 80.1827,Y 115.4944,Z 180,A 57.0284,B 5.0803,C 0.1212,E1 5.1734,E2 395.7828} C_DIS
LIN {X 76.4559,Y 117.9945,Z 180,A 58.8647,B 5.0803,C 0.1182,E1 5.1691,E2 393.9453} C_DIS
LIN {X 72.832,Y 120.2651,Z 180,A 60.541,B 5.0803,C 0.1164,E1 5.1651,E2 392.2776} C_DIS
LIN {X 69.2009,Y 122.391,Z 180,A 62.2976,B 5.0804,C 0.1134,E1 5.1609,E2 390.5157} C_DIS
LIN {X 65.1043,Y 124.6159,Z 180,A 64.0739,B 5.0804,C 0.1124,E1 5.1565,E2 388.7551} C_DIS
LIN {X 62.6706,Y 125.8582,Z 180,A 65.3758,B 5.0805,C 0.1085,E1 5.1532,E2 387.4293} C_DIS
LIN {X 58.5582,Y 127.8234,Z 180,A 66.9509,B 5.0805,C 0.1098,E1 5.1493,E2 385.8904} C_DIS
LIN {X 55.0475,Y 129.3757,Z 180,A 68.5539,B 5.0805,C 0.1075,E1 5.1452,E2 384.2827} C_DIS
LIN {X 52.2827,Y 130.5154,Z 180,A 69.7333,B 5.0805,C 0.1067,E1 5.1422,E2 383.1084} C_DIS
LIN {X 49.1471,Y 131.7279,Z 180,A 71.0864,B 5.0805,C 0.1054,E1 5.1386,E2 381.7576} C_DIS
LIN {X 45.6964,Y 132.9648,Z 180,A 72.5918,B 5.0806,C 0.1038,E1 5.1347,E2 380.2511} C_DIS
LIN {X 41.7929,Y 134.2441,Z 180,A 74.1537,B 5.0806,C 0.1037,E1 5.1305,E2 378.7037} C_DIS
LIN {X 39.1988,Y 135.0231,Z 180,A 75.3286,B 5.0806,C 0.1019,E1 5.1274,E2 377.52} C_DIS
LIN {X 35.7333,Y 135.9819,Z 180,A 77.2975,B 5.0808,C 0.0946,E1 5.1219,E2 375.4872} C_DIS
LIN {X 31.2437,Y 137.0822,Z 180,A 78.6659,B 5.0808,C 0.0995,E1 5.1183,E2 374.1851} C_DIS
LIN {X 27.3401,Y 137.9157,Z 180,A 80.2469,B 5.0808,C 0.0991,E1 5.114,E2 372.6104} C_DIS
LIN {X 24.1455,Y 138.5104,Z 180,A 81.5607,B 5.0808,C 0.0985,E1 5.1104,E2 371.2984} C_DIS
LIN {X 18.3879,Y 139.3902,Z 180,A 83.9787,B 5.0808,C 0.0969,E1 5.1037,E2 368.8754} C_DIS
LIN {X 14.7058,Y 139.8271,Z 180,A 85.4223,B 5.0808,C 0.0971,E1 5.0997,E2 367.4409} C_DIS
LIN {X 11.2322,Y 140.1498,Z 180,A 86.9944,B 5.0808,C 0.095,E1 5.0953,E2 365.8503} C_DIS
LIN {X 7.0252,Y 140.4223,Z 180,A 88.5511,B 5.0808,C 0.0964,E1 5.091,E2 364.3147} C_DIS
LIN {X 3.3641,Y 140.5588,Z 180,A 90.1671,B 5.0808,C 0.0948,E1 5.0865,E2 362.6838} C_DIS
LIN {X -0.8942,Y 140.5952,Z 180,A 91.8332,B 5.0808,C 0.0955,E1 5.0818,E2 361.0272} C_DIS
LIN {X -5.3107,Y 140.4977,Z 180,A 93.6014,B 5.0808,C 0.096,E1 5.0769,E2 359.2639} C_DIS
LIN {X -12.0498,Y 140.0807,Z 180,A 96.3471,B 5.0808,C 0.0964,E1 5.0693,E2 356.5204} C_DIS
LIN {X -15.8044,Y 139.7088,Z 180,A 97.9776,B 5.0808,C 0.0958,E1 5.0647,E2 354.879} C_DIS
LIN {X -19.564,Y 139.2304,Z 180,A 99.89,B 5.0808,C 0.0923,E1 5.0593,E2 352.9205} C_DIS
LIN {X -23.6986,Y 138.5868,Z 180,A 101.287,B 5.0808,C 0.0964,E1 5.0556,E2 351.5637} C_DIS
LIN {X -30.3153,Y 137.2921,Z 180,A 103.7163,B 5.0807,C 0.1012,E1 5.049,E2 349.1763} C_DIS
LIN {X -35.532,Y 136.0356,Z 180,A 106.4014,B 5.0807,C 0.0973,E1 5.0416,E2 346.4295} C_DIS
LIN {X -38.718,Y 135.1639,Z 180,A 107.4632,B 5.0807,C 0.1013,E1 5.0388,E2 345.4046} C_DIS
LIN {X -41.3279,Y 134.3864,Z 180,A 108.5765,B 5.0807,C 0.1021,E1 5.0358,E2 344.2915} C_DIS
LIN {X -44.954,Y 133.2183,Z 180,A 110.1522,B 5.0807,C 0.1032,E1 5.0317,E2 342.7138} C_DIS
LIN {X -48.3603,Y 132.0206,Z 180,A 112.1394,B 5.0807,C 0.0993,E1 5.0263,E2 340.662} C_DIS
LIN {X -52.3792,Y 130.4765,Z 180,A 113.515,B 5.0807,C 0.1049,E1 5.0228,E2 339.3359} C_DIS
LIN {X -56.0935,Y 128.9235,Z 180,A 115.1011,B 5.0806,C 0.1072,E1 5.0188,E2 337.7578} C_DIS
LIN {X -60.0861,Y 127.1127,Z 180,A 117.1251,B 5.0806,C 0.1069,E1 5.0136,E2 335.705} C_DIS
LIN {X -63.874,Y 125.2507,Z 180,A 118.6393,B 5.0805,C 0.1111,E1 5.0099,E2 334.2181} C_DIS
LIN {X -67.1694,Y 123.5172,Z 180,A 120.2543,B 5.0805,C 0.1121,E1 5.0059,E2 332.592} C_DIS
LIN {X -71.1293,Y 121.2799,Z 180,A 122.0211,B 5.0804,C 0.1156,E1 5.0016,E2 330.8376} C_DIS
LIN {X -74.3481,Y 119.3339,Z 180,A 123.6902,B 5.0804,C 0.1165,E1 4.9976,E2 329.1523} C_DIS
LIN {X -78.2381,Y 116.8205,Z 180,A 125.6074,B 5.0803,C 0.1191,E1 4.9931,E2 327.2328} C_DIS
LIN {X -82.3109,Y 113.9876,Z 180,A 128.0028,B 5.0803,C 0.1188,E1 4.9876,E2 324.7913} C_DIS
LIN {X -85.5671,Y 111.5639,Z 180,A 129.4569,B 5.0802,C 0.1235,E1 4.9844,E2 323.3641} C_DIS
LIN {X -89.6309,Y 108.3259,Z 180,A 131.2884,B 5.08,C 0.1299,E1 4.9805,E2 321.5707} C_DIS
LIN {X -94.2556,Y 104.3269,Z 180,A 133.9805,B 5.08,C 0.1327,E1 4.9748,E2 318.8552} C_DIS
LIN {X -99.9238,Y 98.9115,Z 180,A 137.0353,B 5.0798,C 0.1402,E1 4.9687,E2 315.821} C_DIS
LIN {X -103.0348,Y 95.666,Z 180,A 139.3366,B 5.0798,C 0.1397,E1 4.9642,E2 313.4614} C_DIS
LIN {X -108.336,Y 89.6187,Z 180,A 142.0837,B 5.0794,C 0.1515,E1 4.9593,E2 310.7848} C_DIS
LIN {X -111.8521,Y 85.1896,Z 180,A 144.8988,B 5.0794,C 0.1521,E1 4.9543,E2 307.9067} C_DIS
LIN {X -114.0952,Y 82.1625,Z 180,A 146.4532,B 5.0794,C 0.1555,E1 4.9517,E2 306.3512} C_DIS
LIN {X -116.681,Y 78.447,Z 180,A 148.3601,B 5.0792,C 0.1592,E1 4.9487,E2 304.4379} C_DIS
LIN {X -119.1444,Y 74.6525,Z 180,A 150.2391,B 5.0791,C 0.1633,E1 4.9459,E2 302.5559} C_DIS
LIN {X -121.4296,Y 70.8746,Z 180,A 152.087,B 5.0789,C 0.1673,E1 4.9433,E2 300.7033} C_DIS
LIN {X -123.666,Y 66.896,Z 180,A 154.643,B 5.0789,C 0.1659,E1 4.9398,E2 298.0592} C_DIS
LIN {X -126.2711,Y 61.8336,Z 180,A 156.001,B 5.0785,C 0.1801,E1 4.9382,E2 296.8271} C_DIS
LIN {X -127.8604,Y 58.4781,Z 180,A 157.8712,B 5.0785,C 0.1809,E1 4.9359,E2 294.9125} C_DIS
LIN {X -129.4878,Y 54.7811,Z 180,A 160.0275,B 5.0785,C 0.1809,E1 4.9335,E2 292.6917} C_DIS
LIN {X -131.1449,Y 50.6829,Z 180,A 161.0667,B 5.0781,C 0.1921,E1 4.9326,E2 291.7523} C_DIS
LIN {X -132.1188,Y 48.088,Z 180,A 162.6709,B 5.0781,C 0.1911,E1 4.9309,E2 290.0881} C_DIS
LIN {X -133.5065,Y 44.0887,Z 180,A 164.309,B 5.0779,C 0.1965,E1 4.9295,E2 288.4627} C_DIS
LIN {X -134.7869,Y 40.0056,Z 180,A 166.1733,B 5.0778,C 0.2003,E1 4.9279,E2 286.5844} C_DIS
LIN {X -135.9276,Y 35.9369,Z 180,A 167.8805,B 5.0776,C 0.2051,E1 4.9267,E2 284.8805} C_DIS
LIN {X -136.8159,Y 32.395,Z 180,A 169.3873,B 5.0774,C 0.2091,E1 4.9257,E2 283.3725} C_DIS
LIN {X -137.5175,Y 29.2712,Z 180,A 170.806,B 5.0773,C 0.2118,E1 4.9248,E2 281.9401} C_DIS
LIN {X -138.6688,Y 23.2101,Z 180,A 173.3646,B 5.077,C 0.2184,E1 4.9236,E2 279.3778} C_DIS
LIN {X -139.359,Y 18.6263,Z 180,A 175.0771,B 5.0767,C 0.2252,E1 4.9229,E2 277.6897} C_DIS
LIN {X -139.8414,Y 14.5681,Z 180,A 177.212,B 5.0767,C 0.226,E1 4.9222,E2 275.4952} C_DIS
LIN {X -140.2348,Y 10.0993,Z 180,A 178.8665,B 5.0764,C 0.2327,E1 4.9218,E2 273.8647} C_DIS
LIN {X -140.4418,Y 6.6381,Z 180,A -179.5895,B 5.0762,C 0.2356,E1 4.9216,E2 272.3048} C_DIS
LIN {X -140.5762,Y 2.4772,Z 180,A -177.3483,B 5.0762,C 0.2358,E1 4.9216,E2 269.9937} C_DIS
LIN {X -140.5772,Y -2.4181,Z 180,A -175.6026,B 5.0759,C 0.2436,E1 4.9216,E2 268.2821} C_DIS
LIN {X -140.4839,Y -5.6654,Z 180,A -174.1748,B 5.0757,C 0.2465,E1 4.9217,E2 266.8417} C_DIS
LIN {X -140.2859,Y -9.3916,Z 180,A -172.9888,B 5.0754,C 0.2536,E1 4.9219,E2 265.7006} C_DIS
LIN {X -139.9718,Y -13.255,Z 180,A -170.9655,B 5.0754,C 0.2543,E1 4.9225,E2 263.6203} C_DIS
LIN {X -139.5742,Y -16.9369,Z 180,A -169.9344,B 5.0749,C 0.2626,E1 4.9228,E2 262.6528} C_DIS
LIN {X -139.0209,Y -21.0046,Z 180,A -168.1865,B 5.0747,C 0.2667,E1 4.9235,E2 260.8963} C_DIS
LIN {X -138.479,Y -24.3206,Z 180,A -166.4591,B 5.0747,C 0.2675,E1 4.9243,E2 259.123} C_DIS
LIN {X -137.7287,Y -28.2592,Z 180,A -164.9443,B 5.0744,C 0.273,E1 4.9251,E2 257.6248} C_DIS
LIN {X -136.9664,Y -31.751,Z 180,A -163.5006,B 5.0741,C 0.2771,E1 4.926,E2 256.1837} C_DIS
LIN {X -136.1664,Y -35.0228,Z 180,A -161.941,B 5.0741,C 0.2793,E1 4.9271,E2 254.6004} C_DIS
LIN {X -135.0097,Y -39.2446,Z 180,A -160.2004,B 5.0737,C 0.2845,E1 4.9284,E2 252.8666} C_DIS
LIN {X -133.9619,Y -42.6837,Z 180,A -158.6444,B 5.0736,C 0.2877,E1 4.9297,E2 251.2995} C_DIS
LIN {X -132.6752,Y -46.5317,Z 180,A -156.1908,B 5.0737,C 0.2851,E1 4.9321,E2 248.7407} C_DIS
LIN {X -130.5076,Y -52.302,Z 180,A -154.3062,B 5.073,C 0.2972,E1 4.9339,E2 246.9408} C_DIS
LIN {X -129.2736,Y -55.2838,Z 180,A -152.9665,B 5.0728,C 0.3004,E1 4.9354,E2 245.5986} C_DIS
LIN {X -127.4823,Y -59.2958,Z 180,A -151.2726,B 5.0725,C 0.3058,E1 4.9373,E2 243.9183} C_DIS
LIN {X -126.1126,Y -62.155,Z 180,A -149.9466,B 5.0723,C 0.3087,E1 4.9389,E2 242.5885} C_DIS
LIN {X -124.6104,Y -65.1148,Z 180,A -147.0595,B 5.073,C 0.2982,E1 4.9431,E2 239.4966} C_DIS
LIN {X -119.7834,Y -73.6216,Z 180,A -144.8152,B 5.0714,C 0.3237,E1 4.9459,E2 237.4873} C_DIS
LIN {X -117.7282,Y -76.8661,Z 180,A -142.7884,B 5.0714,C 0.3232,E1 4.949,E2 235.4001} C_DIS
LIN {X -115.2797,Y -80.4912,Z 180,A -140.9211,B 5.0712,C 0.3265,E1 4.952,E2 233.5222} C_DIS
LIN {X -112.4552,Y -84.3928,Z 180,A -138.9555,B 5.0709,C 0.3308,E1 4.9552,E2 231.5568} C_DIS
LIN {X -109.9949,Y -87.5746,Z 180,A -137.2906,B 5.0707,C 0.3342,E1 4.9581,E2 229.8891} C_DIS
LIN {X -107.3342,Y -90.8167,Z 180,A -135.4698,B 5.0705,C 0.3367,E1 4.9614,E2 228.0539} C_DIS
LIN {X -104.2912,Y -94.2952,Z 180,A -133.5658,B 5.0703,C 0.3404,E1 4.9649,E2 226.1476} C_DIS
LIN {X -101.1898,Y -97.616,Z 180,A -131.6643,B 5.0701,C 0.3436,E1 4.9686,E2 224.2398} C_DIS
LIN {X -97.9719,Y -100.8452,Z 180,A -129.7666,B 5.0699,C 0.3468,E1 4.9724,E2 222.3372} C_DIS
LIN {X -94.576,Y -104.0364,Z 180,A -127.8562,B 5.0696,C 0.3502,E1 4.9763,E2 220.4255} C_DIS
LIN {X -91.2135,Y -106.9969,Z 180,A -125.9795,B 5.0694,C 0.3529,E1 4.9803,E2 218.5423} C_DIS
LIN {X -87.5822,Y -109.9889,Z 180,A -124.0559,B 5.0692,C 0.3561,E1 4.9844,E2 216.6181} C_DIS
LIN {X -81.7167,Y -114.4141,Z 180,A -121.0455,B 5.0689,C 0.3608,E1 4.9912,E2 213.6059} C_DIS
LIN {X -78.2219,Y -116.8314,Z 180,A -119.2304,B 5.0688,C 0.3625,E1 4.9954,E2 211.7796} C_DIS
LIN {X -74.0248,Y -119.535,Z 180,A -117.1892,B 5.0686,C 0.3654,E1 5.0002,E2 209.7375} C_DIS
LIN {X -70.082,Y -121.8888,Z 180,A -115.2577,B 5.0684,C 0.3672,E1 5.0049,E2 207.798} C_DIS
LIN {X -66.3615,Y -123.9532,Z 180,A -113.693,B 5.0681,C 0.3712,E1 5.0087,E2 206.2559} C_DIS
LIN {X -62.6898,Y -125.8488,Z 180,A -112.0369,B 5.068,C 0.3735,E1 5.0128,E2 204.6033} C_DIS
LIN {X -60.2147,Y -127.0512,Z 180,A -110.7801,B 5.068,C 0.3733,E1 5.016,E2 203.3282} C_DIS
LIN {X -56.4456,Y -128.7713,Z 180,A -109.138,B 5.0678,C 0.3756,E1 5.0202,E2 201.6922} C_DIS
LIN {X -53.9981,Y -129.8148,Z 180,A -107.9917,B 5.0678,C 0.376,E1 5.0232,E2 200.5374} C_DIS
LIN {X -50.3043,Y -131.292,Z 180,A -106.3562,B 5.0677,C 0.3773,E1 5.0274,E2 198.8998} C_DIS
LIN {X -47.5585,Y -132.3097,Z 180,A -104.7074,B 5.068,C 0.3733,E1 5.0319,E2 197.1892} C_DIS
LIN {X -43.5094,Y -133.6981,Z 180,A -103.4245,B 5.0675,C 0.3798,E1 5.0352,E2 195.9683} C_DIS
LIN {X -39.1834,Y -135.0276,Z 180,A -101.1221,B 5.0678,C 0.3759,E1 5.0415,E2 193.6036} C_DIS
LIN {X -35.2533,Y -136.1079,Z 180,A -99.9228,B 5.0673,C 0.3821,E1 5.0446,E2 192.4663} C_DIS
LIN {X -31.197,Y -137.0929,Z 180,A -98.1009,B 5.0673,C 0.3817,E1 5.0496,E2 190.6276} C_DIS
LIN {X -27.2537,Y -137.9333,Z 180,A -96.5113,B 5.0673,C 0.383,E1 5.0539,E2 189.0447} C_DIS
LIN {X -23.5757,Y -138.6078,Z 180,A -94.929,B 5.0673,C 0.383,E1 5.0583,E2 187.454} C_DIS
LIN {X -19.9428,Y -139.1762,Z 180,A -93.4495,B 5.0673,C 0.3836,E1 5.0624,E2 185.9766} C_DIS
LIN {X -15.8682,Y -139.7017,Z 180,A -91.6572,B 5.0673,C 0.3825,E1 5.0674,E2 184.1677} C_DIS
LIN {X -11.7995,Y -140.1019,Z 180,A -90.1346,B 5.0672,C 0.3844,E1 5.0716,E2 182.6638} C_DIS
LIN {X -8.5373,Y -140.3385,Z 180,A -88.7801,B 5.0672,C 0.3843,E1 5.0753,E2 181.3058} C_DIS
LIN {X -4.4766,Y -140.5278,Z 180,A -87.0496,B 5.0672,C 0.3834,E1 5.0802,E2 179.5647} C_DIS
LIN {X -0.5038,Y -140.5974,Z 180,A -85.4655,B 5.0672,C 0.3836,E1 5.0846,E2 177.9845} C_DIS
LIN {X -0.5038,Y -140.5974,Z 180,A -85.4655,B 5.0672,C 0.3836,E1 5.0846,E2 177.9845} C_DIS
Enddeposition()
LIN {X 0.9938,Y -141.4962,Z 180,A -85.3901,B 5.0654,C 0.3928,E1 5.0835,E2 178.0134} C_DIS
Startdeposition()
$VEL.CP = VEL_PRINT
LIN {X -1.5547,Y -141.4942,Z 180,A -86.5632,B 5.0654,C 0.3946,E1 5.0801,E2 179.2061} C_DIS
LIN {X -4.8865,Y -141.4176,Z 180,A -87.9825,B 5.0652,C 0.3955,E1 5.0761,E2 180.6355} C_DIS
LIN {X -9.3289,Y -141.1941,Z 180,A -89.6713,B 5.0653,C 0.3941,E1 5.0715,E2 182.3099} C_DIS
LIN {X -12.6355,Y -140.9371,Z 180,A -91.1628,B 5.0653,C 0.3957,E1 5.0673,E2 183.822} C_DIS
LIN {X -17.2071,Y -140.4511,Z 180,A -93.0182,B 5.0653,C 0.3952,E1 5.0621,E2 185.6772} C_DIS
LIN {X -21.7359,Y -139.8211,Z 180,A -94.7658,B 5.0653,C 0.3935,E1 5.0573,E2 187.4114} C_DIS
LIN {X -25.3616,Y -139.2097,Z 180,A -96.2943,B 5.0653,C 0.3935,E1 5.0531,E2 188.9458} C_DIS
LIN {X -29.2086,Y -138.4545,Z 180,A -97.9705,B 5.0653,C 0.3937,E1 5.0485,E2 190.6345} C_DIS
LIN {X -33.0856,Y -137.5779,Z 180,A -99.4456,B 5.0656,C 0.3914,E1 5.0445,E2 192.0919} C_DIS
LIN {X -36.1199,Y -136.813,Z 180,A -100.6443,B 5.0656,C 0.3899,E1 5.0413,E2 193.2817} C_DIS
LIN {X -38.4501,Y -136.1765,Z 180,A -101.8218,B 5.0656,C 0.3915,E1 5.0381,E2 194.4863} C_DIS
LIN {X -42.2166,Y -135.0584,Z 180,A -103.3587,B 5.0656,C 0.3897,E1 5.034,E2 196.0164} C_DIS
LIN {X -47.4686,Y -133.3017,Z 180,A -105.9488,B 5.0656,C 0.3917,E1 5.027,E2 198.6534} C_DIS
LIN {X -51.0011,Y -131.9896,Z 180,A -107.0415,B 5.066,C 0.3857,E1 5.0243,E2 199.6884} C_DIS
LIN {X -53.8176,Y -130.8684,Z 180,A -108.4475,B 5.066,C 0.3864,E1 5.0206,E2 201.1185} C_DIS
LIN {X -57.4276,Y -129.3232,Z 180,A -109.9613,B 5.0661,C 0.384,E1 5.0167,E2 202.6224} C_DIS
LIN {X -60.8218,Y -127.7615,Z 180,A -111.5339,B 5.0662,C 0.383,E1 5.0127,E2 204.203} C_DIS
LIN {X -64.0423,Y -126.178,Z 180,A -113.0667,B 5.0662,C 0.3821,E1 5.0089,E2 205.7467} C_DIS
LIN {X -66.9389,Y -124.6677,Z 180,A -114.6154,B 5.0662,C 0.3828,E1 5.005,E2 207.3257} C_DIS
LIN {X -70.0084,Y -122.9703,Z 180,A -115.7976,B 5.0665,C 0.3785,E1 5.0022,E2 208.4762} C_DIS
LIN {X -73.7153,Y -120.785,Z 180,A -117.6215,B 5.0666,C 0.377,E1 4.9978,E2 210.311} C_DIS
LIN {X -77.5922,Y -118.3316,Z 180,A -119.5031,B 5.0668,C 0.3746,E1 4.9934,E2 212.1957} C_DIS
LIN {X -81.4392,Y -115.7174,Z 180,A -121.3904,B 5.067,C 0.3717,E1 4.989,E2 214.0835} C_DIS
LIN {X -84.3772,Y -113.5929,Z 180,A -122.9427,B 5.0671,C 0.3702,E1 4.9855,E2 215.647} C_DIS
LIN {X -88.3516,Y -110.5302,Z 180,A -124.9293,B 5.0674,C 0.3664,E1 4.9812,E2 217.6274} C_DIS
LIN {X -91.7671,Y -107.711,Z 180,A -126.7213,B 5.0676,C 0.3633,E1 4.9773,E2 219.4189} C_DIS
LIN {X -94.9719,Y -104.8961,Z 180,A -128.5482,B 5.0678,C 0.3611,E1 4.9735,E2 221.2588} C_DIS
LIN {X -98.4098,Y -101.6777,Z 180,A -130.4729,B 5.068,C 0.3577,E1 4.9696,E2 223.1855} C_DIS
LIN {X -101.7285,Y -98.3573,Z 180,A -132.3527,B 5.0683,C 0.3538,E1 4.9659,E2 225.0621} C_DIS
LIN {X -104.5177,Y -95.3889,Z 180,A -134.0687,B 5.0685,C 0.3511,E1 4.9626,E2 226.7866} C_DIS
LIN {X -107.4185,Y -92.1097,Z 180,A -135.9102,B 5.0687,C 0.3481,E1 4.9592,E2 228.6367} C_DIS
LIN {X -110.316,Y -88.6188,Z 180,A -137.7787,B 5.069,C 0.3444,E1 4.9559,E2 230.5089} C_DIS
LIN {X -112.9355,Y -85.255,Z 180,A -139.544,B 5.0692,C 0.341,E1 4.9529,E2 232.2788} C_DIS
LIN {X -115.689,Y -81.4795,Z 180,A -141.4928,B 5.0694,C 0.3373,E1 4.9497,E2 234.2344} C_DIS
LIN {X -118.3435,Y -77.5741,Z 180,A -143.5009,B 5.0697,C 0.3337,E1 4.9466,E2 236.2545} C_DIS
LIN {X -120.9081,Y -73.5131,Z 180,A -145.4686,B 5.07,C 0.3293,E1 4.9437,E2 238.2245} C_DIS
LIN {X -123.0942,Y -69.7911,Z 180,A -147.7099,B 5.07,C 0.3295,E1 4.9405,E2 240.5298} C_DIS
LIN {X -125.3497,Y -65.6485,Z 180,A -149.0579,B 5.0706,C 0.3198,E1 4.9389,E2 241.8031} C_DIS
LIN {X -126.8279,Y -62.7454,Z 180,A -150.4248,B 5.0708,C 0.3169,E1 4.9371,E2 243.1757} C_DIS
LIN {X -128.5328,Y -59.1746,Z 180,A -152.2178,B 5.0708,C 0.3145,E1 4.935,E2 244.9931} C_DIS
LIN {X -130.4441,Y -54.8337,Z 180,A -153.9686,B 5.0713,C 0.3081,E1 4.9331,E2 246.7206} C_DIS
LIN {X -131.3084,Y -52.7296,Z 180,A -155.7866,B 5.071,C 0.3134,E1 4.9311,E2 248.6553} C_DIS
LIN {X -133.4455,Y -47.0657,Z 180,A -157.6227,B 5.0717,C 0.3017,E1 4.9294,E2 250.41} C_DIS
LIN {X -134.7349,Y -43.2301,Z 180,A -159.2843,B 5.0719,C 0.2975,E1 4.928,E2 252.0737} C_DIS
LIN {X -136.0449,Y -38.9207,Z 180,A -161.2136,B 5.0722,C 0.2934,E1 4.9264,E2 254.0158} C_DIS
LIN {X -137.0876,Y -35.0627,Z 180,A -162.7354,B 5.0725,C 0.2882,E1 4.9253,E2 255.5238} C_DIS
LIN {X -137.8626,Y -31.8807,Z 180,A -164.1005,B 5.0726,C 0.2849,E1 4.9245,E2 256.8933} C_DIS
LIN {X -138.5598,Y -28.7015,Z 180,A -165.3763,B 5.0729,C 0.2809,E1 4.9237,E2 258.1627} C_DIS
LIN {X -139.4364,Y -24.0938,Z 180,A -167.6018,B 5.073,C 0.2783,E1 4.9226,E2 260.4297} C_DIS
LIN {X -140.3276,Y -18.182,Z 180,A -169.9593,B 5.0734,C 0.271,E1 4.9217,E2 262.7771} C_DIS
LIN {X -140.9709,Y -12.2356,Z 180,A -172.4463,B 5.0737,C 0.2647,E1 4.921,E2 265.271} C_DIS
LIN {X -141.2386,Y -8.6069,Z 180,A -173.9515,B 5.0739,C 0.2608,E1 4.9207,E2 266.7793} C_DIS
LIN {X -141.4353,Y -4.3159,Z 180,A -175.956,B 5.0741,C 0.2581,E1 4.9205,E2 268.8168} C_DIS
LIN {X -141.4964,Y 1.236,Z 180,A -178.1539,B 5.0744,C 0.2513,E1 4.9205,E2 271.0066} C_DIS
LIN {X -141.4137,Y 4.9858,Z 180,A -179.6848,B 5.0746,C 0.2471,E1 4.9205,E2 272.538} C_DIS
LIN {X -141.1789,Y 9.5636,Z 180,A 178.3462,B 5.0748,C 0.2427,E1 4.9209,E2 274.5202} C_DIS
LIN {X -140.8383,Y 13.6748,Z 180,A 176.4394,B 5.075,C 0.24,E1 4.9214,E2 276.456} C_DIS
LIN {X -140.4388,Y 17.3101,Z 180,A 175.1532,B 5.0752,C 0.2342,E1 4.9218,E2 277.716} C_DIS
LIN {X -139.9423,Y 20.9531,Z 180,A 173.6548,B 5.0754,C 0.2301,E1 4.9224,E2 279.2145} C_DIS
LIN {X -139.4998,Y 23.714,Z 180,A 171.814,B 5.0753,C 0.2327,E1 4.9234,E2 281.1451} C_DIS
LIN {X -138.4169,Y 29.3827,Z 180,A 170.1151,B 5.0758,C 0.2209,E1 4.9243,E2 282.7606} C_DIS
LIN {X -137.6004,Y 32.9924,Z 180,A 168.6826,B 5.076,C 0.2162,E1 4.9252,E2 284.1833} C_DIS
LIN {X -136.8125,Y 36.1221,Z 180,A 167.3263,B 5.0762,C 0.213,E1 4.9261,E2 285.5449} C_DIS
LIN {X -136.0134,Y 39.0289,Z 180,A 166.0543,B 5.0762,C 0.2101,E1 4.9271,E2 286.8225} C_DIS
LIN {X -134.8928,Y 42.7357,Z 180,A 164.4044,B 5.0764,C 0.2065,E1 4.9284,E2 288.4816} C_DIS
LIN {X -133.8119,Y 46.0087,Z 180,A 163.1076,B 5.0766,C 0.2019,E1 4.9296,E2 289.7645} C_DIS
LIN {X -132.5453,Y 49.5382,Z 180,A 161.5176,B 5.0767,C 0.1985,E1 4.9311,E2 291.3625} C_DIS
LIN {X -131.687,Y 51.7796,Z 180,A 160.0755,B 5.0767,C 0.1999,E1 4.9326,E2 292.8639} C_DIS
LIN {X -130.3458,Y 55.0689,Z 180,A 158.8446,B 5.0769,C 0.1944,E1 4.9339,E2 294.0671} C_DIS
LIN {X -128.6366,Y 58.9503,Z 180,A 157.1201,B 5.0771,C 0.19,E1 4.9359,E2 295.7912} C_DIS
LIN {X -127.449,Y 61.4759,Z 180,A 155.6776,B 5.0771,C 0.1897,E1 4.9377,E2 297.2725} C_DIS
LIN {X -125.8837,Y 64.6204,Z 180,A 154.3247,B 5.0772,C 0.1855,E1 4.9394,E2 298.6153} C_DIS
LIN {X -123.4265,Y 69.201,Z 180,A 152.3018,B 5.0774,C 0.1796,E1 4.9421,E2 300.6261} C_DIS
LIN {X -121.1789,Y 73.0654,Z 180,A 150.4239,B 5.0776,C 0.1758,E1 4.9448,E2 302.511} C_DIS
LIN {X -118.6924,Y 77.0386,Z 180,A 148.5142,B 5.0777,C 0.1713,E1 4.9476,E2 304.4206} C_DIS
LIN {X -116.3843,Y 80.4842,Z 180,A 146.7532,B 5.0778,C 0.1681,E1 4.9504,E2 306.1905} C_DIS
LIN {X -114.3371,Y 83.3669,Z 180,A 144.6192,B 5.0778,C 0.1709,E1 4.9541,E2 308.412} C_DIS
LIN {X -110.7178,Y 88.1158,Z 180,A 142.8763,B 5.0781,C 0.1596,E1 4.9569,E2 310.0678} C_DIS
LIN {X -106.3908,Y 93.295,Z 180,A 139.9005,B 5.0782,C 0.1559,E1 4.9624,E2 313.0721} C_DIS
LIN {X -101.6864,Y 98.4008,Z 180,A 137.2182,B 5.0784,C 0.149,E1 4.9675,E2 315.7357} C_DIS
LIN {X -98.8309,Y 101.269,Z 180,A 135.5159,B 5.0785,C 0.1463,E1 4.9708,E2 317.4447} C_DIS
LIN {X -96.0739,Y 103.8885,Z 180,A 133.8735,B 5.0785,C 0.1443,E1 4.9742,E2 319.0988} C_DIS
LIN {X -91.2346,Y 108.163,Z 180,A 131.2319,B 5.0787,C 0.1397,E1 4.9798,E2 321.7417} C_DIS
LIN {X -87.7379,Y 111.0183,Z 180,A 129.4117,B 5.0787,C 0.1364,E1 4.9838,E2 323.5595} C_DIS
LIN {X -80.4708,Y 116.3935,Z 180,A 125.6539,B 5.0789,C 0.1313,E1 4.9923,E2 327.3267} C_DIS
LIN {X -76.616,Y 118.9663,Z 180,A 123.8083,B 5.079,C 0.1282,E1 4.9966,E2 329.1671} C_DIS
LIN {X -73.6942,Y 120.7979,Z 180,A 122.368,B 5.079,C 0.1265,E1 5,E2 330.6118} C_DIS
LIN {X -69.5207,Y 123.2467,Z 180,A 120.4013,B 5.0791,C 0.1239,E1 5.0048,E2 332.578} C_DIS
LIN {X -65.9705,Y 125.1807,Z 180,A 118.8334,B 5.0791,C 0.1211,E1 5.0086,E2 334.1359} C_DIS
LIN {X -62.4176,Y 126.9896,Z 180,A 117.1924,B 5.0792,C 0.1193,E1 5.0127,E2 335.7791} C_DIS
LIN {X -59.2442,Y 128.5007,Z 180,A 115.7272,B 5.0792,C 0.1181,E1 5.0164,E2 337.2486} C_DIS
LIN {X -56.2328,Y 129.8467,Z 180,A 114.5088,B 5.0793,C 0.1154,E1 5.0195,E2 338.4513} C_DIS
LIN {X -52.8778,Y 131.2487,Z 180,A 112.897,B 5.0793,C 0.1153,E1 5.0237,E2 340.0796} C_DIS
LIN {X -47.8613,Y 133.1601,Z 180,A 110.7285,B 5.0793,C 0.1132,E1 5.0294,E2 342.2461} C_DIS
LIN {X -45.2057,Y 134.0859,Z 180,A 109.6742,B 5.0794,C 0.1113,E1 5.0321,E2 343.2889} C_DIS
LIN {X -41.7215,Y 135.21,Z 180,A 107.9498,B 5.0794,C 0.1126,E1 5.0368,E2 345.043} C_DIS
LIN {X -34.7661,Y 137.1629,Z 180,A 105.0532,B 5.0794,C 0.1102,E1 5.0446,E2 347.9341} C_DIS
LIN {X -30.4771,Y 138.1807,Z 180,A 103.3823,B 5.0794,C 0.108,E1 5.0491,E2 349.5897} C_DIS
LIN {X -27.863,Y 138.7304,Z 180,A 102.2683,B 5.0794,C 0.1077,E1 5.0521,E2 350.7071} C_DIS
LIN {X -22.1091,Y 139.7631,Z 180,A 99.7491,B 5.0794,C 0.1083,E1 5.0591,E2 353.2441} C_DIS
LIN {X -18.7822,Y 140.249,Z 180,A 98.5899,B 5.0795,C 0.1057,E1 5.0623,E2 354.3771} C_DIS
LIN {X -16.0722,Y 140.5865,Z 180,A 97.4013,B 5.0795,C 0.1063,E1 5.0656,E2 355.5757} C_DIS
LIN {X -13.3196,Y 140.8724,Z 180,A 96.3049,B 5.0795,C 0.1057,E1 5.0686,E2 356.6684} C_DIS
LIN {X -9.3393,Y 141.1934,Z 180,A 94.4249,B 5.0795,C 0.1084,E1 5.0739,E2 358.5809} C_DIS
LIN {X -4.8375,Y 141.4195,Z 180,A 92.8081,B 5.0795,C 0.1059,E1 5.0784,E2 360.1705} C_DIS
LIN {X -0.6922,Y 141.499,Z 180,A 91.1334,B 5.0795,C 0.1059,E1 5.0831,E2 361.844} C_DIS
LIN {X 2.7755,Y 141.4741,Z 180,A 89.5948,B 5.0795,C 0.1075,E1 5.0874,E2 363.3989} C_DIS
LIN {X 7.0066,Y 141.3271,Z 180,A 87.979,B 5.0795,C 0.1067,E1 5.0919,E2 365.0015} C_DIS
LIN {X 10.6402,Y 141.1004,Z 180,A 86.4468,B 5.0795,C 0.1077,E1 5.0962,E2 366.5406} C_DIS
LIN {X 14.9105,Y 140.7129,Z 180,A 84.8762,B 5.0795,C 0.1064,E1 5.1005,E2 368.0896} C_DIS
LIN {X 17.7944,Y 140.3784,Z 180,A 83.5552,B 5.0795,C 0.1085,E1 5.1042,E2 369.4286} C_DIS
LIN {X 22.5635,Y 139.6918,Z 180,A 81.6444,B 5.0795,C 0.109,E1 5.1094,E2 371.3337} C_DIS
LIN {X 26.4444,Y 139.0074,Z 180,A 80.1434,B 5.0795,C 0.1088,E1 5.1135,E2 372.8222} C_DIS
LIN {X 29.2856,Y 138.4379,Z 180,A 79.0435,B 5.0795,C 0.1086,E1 5.1165,E2 373.9125} C_DIS
LIN {X 32.5681,Y 137.7027,Z 180,A 77.684,B 5.0795,C 0.1095,E1 5.1202,E2 375.2714} C_DIS
LIN {X 36.9087,Y 136.6027,Z 180,A 75.654,B 5.0794,C 0.1135,E1 5.1258,E2 377.3283} C_DIS
LIN {X 42.596,Y 134.9375,Z 180,A 73.3628,B 5.0794,C 0.1142,E1 5.1319,E2 379.6053} C_DIS
LIN {X 47.721,Y 133.2107,Z 180,A 71.3013,B 5.0794,C 0.1148,E1 5.1373,E2 381.6501} C_DIS
LIN {X 50.8511,Y 132.0479,Z 180,A 69.8755,B 5.0793,C 0.1171,E1 5.141,E2 383.0851} C_DIS
LIN {X 54.3063,Y 130.6643,Z 180,A 68.3401,B 5.0793,C 0.1191,E1 5.145,E2 384.6239} C_DIS
LIN {X 58.0744,Y 129.0339,Z 180,A 66.7096,B 5.0792,C 0.1207,E1 5.1492,E2 386.2501} C_DIS
LIN {X 61.4523,Y 127.4603,Z 180,A 65.2094,B 5.0792,C 0.1225,E1 5.1529,E2 387.7492} C_DIS
LIN {X 67.3156,Y 124.4653,Z 180,A 62.5976,B 5.0791,C 0.1254,E1 5.1594,E2 390.3541} C_DIS
LIN {X 71.1369,Y 122.3211,Z 180,A 60.8679,B 5.0791,C 0.1274,E1 5.1636,E2 392.078} C_DIS
LIN {X 74.673,Y 120.1948,Z 180,A 59.2142,B 5.079,C 0.1297,E1 5.1675,E2 393.7296} C_DIS
LIN {X 77.9913,Y 118.0688,Z 180,A 57.6056,B 5.0789,C 0.1324,E1 5.1713,E2 395.3399} C_DIS
LIN {X 81.5445,Y 115.6431,Z 180,A 56.0834,B 5.0789,C 0.1324,E1 5.1747,E2 396.8341} C_DIS
LIN {X 84.4665,Y 113.5264,Z 180,A 54.4575,B 5.0788,C 0.137,E1 5.1784,E2 398.4812} C_DIS
LIN {X 88.0512,Y 110.7693,Z 180,A 52.6763,B 5.0788,C 0.1396,E1 5.1823,E2 400.2562} C_DIS
LIN {X 90.1936,Y 109.0319,Z 180,A 51.424,B 5.0786,C 0.1435,E1 5.1851,E2 401.5259} C_DIS
LIN {X 96.0797,Y 103.8832,Z 180,A 47.9405,B 5.0783,C 0.1538,E1 5.1924,E2 405.0502} C_DIS
LIN {X 99.7294,Y 100.3836,Z 180,A 46.468,B 5.0784,C 0.1501,E1 5.1952,E2 406.45} C_DIS
LIN {X 102.7677,Y 97.2712,Z 180,A 44.6836,B 5.0783,C 0.1541,E1 5.1987,E2 408.2377} C_DIS
LIN {X 104.9146,Y 94.9516,Z 180,A 43.3628,B 5.0782,C 0.1574,E1 5.2012,E2 409.5642} C_DIS
LIN {X 111.4512,Y 87.1868,Z 180,A 39.4219,B 5.078,C 0.1641,E1 5.2081,E2 413.4846} C_DIS
LIN {X 114.2167,Y 83.5313,Z 180,A 37.5986,B 5.0778,C 0.1679,E1 5.2112,E2 415.3044} C_DIS
LIN {X 116.8243,Y 79.8436,Z 180,A 35.8459,B 5.0778,C 0.1711,E1 5.2139,E2 417.0479} C_DIS
LIN {X 119.128,Y 76.3634,Z 180,A 34.2443,B 5.0776,C 0.1739,E1 5.2164,E2 418.6388} C_DIS
LIN {X 121.1906,Y 73.0461,Z 180,A 32.68,B 5.0776,C 0.1775,E1 5.2186,E2 420.2015} C_DIS
LIN {X 123.7492,Y 68.6221,Z 180,A 30.6112,B 5.0773,C 0.1826,E1 5.2215,E2 422.271} C_DIS
LIN {X 125.8458,Y 64.6947,Z 180,A 28.8977,B 5.0773,C 0.1859,E1 5.2237,E2 423.9739} C_DIS
LIN {X 127.3783,Y 61.624,Z 180,A 27.5576,B 5.0771,C 0.1887,E1 5.2254,E2 425.3082} C_DIS
LIN {X 129.0096,Y 58.1287,Z 180,A 25.9676,B 5.077,C 0.1932,E1 5.2272,E2 426.9026} C_DIS
LIN {X 130.8582,Y 53.8418,Z 180,A 24.0699,B 5.0768,C 0.1982,E1 5.2293,E2 428.8022} C_DIS
LIN {X 132.7895,Y 48.8864,Z 180,A 22.1065,B 5.0766,C 0.2012,E1 5.2312,E2 430.7422} C_DIS
LIN {X 134.0213,Y 45.3996,Z 180,A 20.5408,B 5.0764,C 0.2062,E1 5.2326,E2 432.3176} C_DIS
LIN {X 135.3605,Y 41.2295,Z 180,A 18.9061,B 5.0764,C 0.209,E1 5.234,E2 433.9352} C_DIS
LIN {X 136.6078,Y 36.8895,Z 180,A 17.0852,B 5.0761,C 0.2139,E1 5.2354,E2 435.7562} C_DIS
LIN {X 137.4756,Y 33.5101,Z 180,A 15.8126,B 5.0761,C 0.2158,E1 5.2362,E2 437.0115} C_DIS
LIN {X 138.1471,Y 30.6327,Z 180,A 14.6517,B 5.0759,C 0.2186,E1 5.2369,E2 438.1685} C_DIS
LIN {X 138.8817,Y 27.1019,Z 180,A 13.317,B 5.0759,C 0.2208,E1 5.2377,E2 439.4877} C_DIS
LIN {X 139.5169,Y 23.6119,Z 180,A 11.7865,B 5.0756,C 0.2262,E1 5.2384,E2 441.0314} C_DIS
LIN {X 140.0039,Y 20.5319,Z 180,A 10.6947,B 5.0756,C 0.2272,E1 5.2389,E2 442.1018} C_DIS
LIN {X 140.6123,Y 15.8458,Z 180,A 8.7714,B 5.0753,C 0.2328,E1 5.2395,E2 444.0278} C_DIS
LIN {X 140.9889,Y 12.0228,Z 180,A 7.1287,B 5.075,C 0.2385,E1 5.24,E2 445.6829} C_DIS
LIN {X 141.3009,Y 7.5274,Z 180,A 5.499,B 5.075,C 0.2408,E1 5.2402,E2 447.2884} C_DIS
LIN {X 141.4429,Y 4.0452,Z 180,A 4.0429,B 5.0747,C 0.2454,E1 5.2404,E2 448.7514} C_DIS
LIN {X 141.5023,Y 0.3592,Z 180,A 2.4704,B 5.0744,C 0.2509,E1 5.2404,E2 450.3355} C_DIS
LIN {X 141.4477,Y -3.8691,Z 180,A 0.9591,B 5.0744,C 0.2528,E1 5.2404,E2 451.8217} C_DIS
LIN {X 141.3473,Y -6.6038,Z 180,A -0.0971,B 5.0742,C 0.2552,E1 5.2402,E2 452.8719} C_DIS
LIN {X 141.144,Y -10.0428,Z 180,A -1.5122,B 5.074,C 0.2594,E1 5.24,E2 454.2908} C_DIS
LIN {X 140.871,Y -13.3339,Z 180,A -2.7215,B 5.074,C 0.2613,E1 5.2397,E2 455.4843} C_DIS
LIN {X 140.5802,Y -16.1249,Z 180,A -3.9369,B 5.0737,C 0.2657,E1 5.2393,E2 456.711} C_DIS
LIN {X 140.0686,Y -20.0789,Z 180,A -5.4907,B 5.0735,C 0.2694,E1 5.2387,E2 458.2581} C_DIS
LIN {X 139.4126,Y -24.2282,Z 180,A -7.0693,B 5.0733,C 0.2724,E1 5.238,E2 459.822} C_DIS
LIN {X 138.5285,Y -28.8554,Z 180,A -8.9804,B 5.073,C 0.2778,E1 5.237,E2 461.7352} C_DIS
LIN {X 137.667,Y -32.7159,Z 180,A -10.6082,B 5.0728,C 0.2826,E1 5.236,E2 463.3677} C_DIS
LIN {X 136.7335,Y -36.4182,Z 180,A -12.0506,B 5.0726,C 0.2854,E1 5.235,E2 464.7977} C_DIS
LIN {X 134.7621,Y -43.1452,Z 180,A -14.8656,B 5.0722,C 0.2928,E1 5.2327,E2 467.612} C_DIS
LIN {X 133.3013,Y -47.4697,Z 180,A -16.7043,B 5.0719,C 0.2977,E1 5.231,E2 469.4511} C_DIS
LIN {X 131.9466,Y -51.1117,Z 180,A -18.0595,B 5.0719,C 0.2987,E1 5.2297,E2 470.7786} C_DIS
LIN {X 130.6519,Y -54.3361,Z 180,A -19.5439,B 5.0716,C 0.3036,E1 5.2281,E2 472.2746} C_DIS
LIN {X 129.1719,Y -57.7658,Z 180,A -20.9459,B 5.0714,C 0.306,E1 5.2266,E2 473.6633} C_DIS
LIN {X 127.9315,Y -60.466,Z 180,A -22.2218,B 5.0712,C 0.3102,E1 5.225,E2 474.9499} C_DIS
LIN {X 126.2838,Y -63.8344,Z 180,A -23.6593,B 5.071,C 0.3129,E1 5.2233,E2 476.3779} C_DIS
LIN {X 124.4528,Y -67.3389,Z 180,A -25.2953,B 5.0707,C 0.3175,E1 5.2211,E2 478.0201} C_DIS
LIN {X 122.2328,Y -71.2893,Z 180,A -26.8391,B 5.0707,C 0.3179,E1 5.219,E2 479.5267} C_DIS
LIN {X 119.9794,Y -75.0192,Z 180,A -28.8081,B 5.0702,C 0.3252,E1 5.2161,E2 481.5245} C_DIS
LIN {X 117.4457,Y -78.9273,Z 180,A -30.6075,B 5.07,C 0.3285,E1 5.2134,E2 483.3141} C_DIS
LIN {X 114.9109,Y -82.5738,Z 180,A -32.2058,B 5.07,C 0.3299,E1 5.2109,E2 484.8873} C_DIS
LIN {X 111.9141,Y -86.5915,Z 180,A -34.4349,B 5.0694,C 0.3375,E1 5.2071,E2 487.1448} C_DIS
LIN {X 109.039,Y -90.185,Z 180,A -36.1834,B 5.0692,C 0.3401,E1 5.204,E2 488.8796} C_DIS
LIN {X 106.3957,Y -93.2894,Z 180,A -37.7916,B 5.069,C 0.3432,E1 5.2011,E2 490.4835} C_DIS
LIN {X 103.428,Y -96.5687,Z 180,A -39.5497,B 5.0688,C 0.3466,E1 5.1977,E2 492.2389} C_DIS
LIN {X 100.3824,Y -99.7307,Z 180,A -41.2631,B 5.0686,C 0.3494,E1 5.1944,E2 493.9452} C_DIS
LIN {X 97.3408,Y -102.7021,Z 180,A -42.9913,B 5.0684,C 0.353,E1 5.1909,E2 495.6758} C_DIS
LIN {X 94.2636,Y -105.5331,Z 180,A -44.6145,B 5.0682,C 0.3554,E1 5.1876,E2 497.291} C_DIS
LIN {X 91.2191,Y -108.1759,Z 180,A -46.2366,B 5.068,C 0.3584,E1 5.1842,E2 498.9131} C_DIS
LIN {X 88.0418,Y -110.7767,Z 180,A -47.8531,B 5.0678,C 0.3609,E1 5.1807,E2 500.5248} C_DIS
LIN {X 84.8589,Y -113.2339,Z 180,A -49.5081,B 5.0676,C 0.3642,E1 5.177,E2 502.1847} C_DIS
LIN {X 81.6507,Y -115.5682,Z 180,A -51.1601,B 5.0673,C 0.3676,E1 5.1732,E2 503.8441} C_DIS
LIN {X 77.589,Y -118.3336,Z 180,A -52.9746,B 5.0673,C 0.3685,E1 5.169,E2 505.6368} C_DIS
LIN {X 74.0148,Y -120.6012,Z 180,A -54.701,B 5.0671,C 0.3715,E1 5.1649,E2 507.3662} C_DIS
LIN {X 71.3517,Y -122.1962,Z 180,A -56.3602,B 5.0665,C 0.3788,E1 5.1608,E2 509.0804} C_DIS
LIN {X 67.3664,Y -124.438,Z 180,A -57.8444,B 5.0667,C 0.3766,E1 5.1573,E2 510.5169} C_DIS
LIN {X 62.982,Y -126.7112,Z 180,A -59.6226,B 5.0667,C 0.3764,E1 5.1529,E2 512.2667} C_DIS
LIN {X 59.8146,Y -128.2369,Z 180,A -61.0716,B 5.0665,C 0.3787,E1 5.1493,E2 513.7202} C_DIS
LIN {X 56.863,Y -129.5742,Z 180,A -62.3531,B 5.0665,C 0.3799,E1 5.146,E2 514.9986} C_DIS
LIN {X 53.1383,Y -131.1437,Z 180,A -63.9904,B 5.0663,C 0.3819,E1 5.1418,E2 516.6371} C_DIS
LIN {X 50.0981,Y -132.3356,Z 180,A -65.203,B 5.0663,C 0.3819,E1 5.1386,E2 517.8359} C_DIS
LIN {X 47.0471,Y -133.4519,Z 180,A -66.6865,B 5.066,C 0.3856,E1 5.1347,E2 519.343} C_DIS
LIN {X 43.3277,Y -134.7038,Z 180,A -68.063,B 5.066,C 0.3844,E1 5.1311,E2 520.6918} C_DIS
LIN {X 38.9909,Y -136.0245,Z 180,A -70.1241,B 5.0657,C 0.389,E1 5.1255,E2 522.7847} C_DIS
LIN {X 34.685,Y -137.1834,Z 180,A -72.243,B 5.0653,C 0.3945,E1 5.1196,E2 524.9467} C_DIS
LIN {X 30.3471,Y -138.2087,Z 180,A -73.6414,B 5.0656,C 0.3907,E1 5.116,E2 526.2917} C_DIS
LIN {X 26.8883,Y -138.9226,Z 180,A -75.0369,B 5.0656,C 0.3913,E1 5.1122,E2 527.6835} C_DIS
LIN {X 22.7141,Y -139.6667,Z 180,A -76.8044,B 5.0654,C 0.3929,E1 5.1073,E2 529.4588} C_DIS
LIN {X 18.094,Y -140.3392,Z 180,A -78.5461,B 5.0655,C 0.3921,E1 5.1025,E2 531.1815} C_DIS
LIN {X 14.1592,Y -140.7918,Z 180,A -80.2446,B 5.0654,C 0.3939,E1 5.0977,E2 532.8937} C_DIS
LIN {X 10.3419,Y -141.1221,Z 180,A -81.5595,B 5.0655,C 0.3916,E1 5.0942,E2 534.1775} C_DIS
LIN {X 7.0948,Y -141.3226,Z 180,A -83.0407,B 5.0654,C 0.394,E1 5.09,E2 535.6814} C_DIS
LIN {X 2.9557,Y -141.4711,Z 180,A -84.6577,B 5.0654,C 0.3936,E1 5.0855,E2 537.2912} C_DIS
LIN {X 2.9557,Y -141.4711,Z 180,A -84.6577,B 5.0654,C 0.3936,E1 5.0855,E2 537.2912} C_DIS
Enddeposition()
LIN {X 1.0001,Y -142.3991,Z 180,A -85.1615,B 5.0656,C 0.3931,E1 5.0843,E2 537.7885} C_DIS
Startdeposition()
$VEL.CP = VEL_PRINT
LIN {X 3.493,Y -142.3612,Z 180,A -83.7616,B 5.066,C 0.388,E1 5.0883,E2 536.3337} C_DIS
LIN {X 7.0021,Y -142.2311,Z 180,A -82.3358,B 5.066,C 0.3875,E1 5.0923,E2 534.9054} C_DIS
LIN {X 12.2245,Y -141.8777,Z 180,A -80.3438,B 5.066,C 0.3882,E1 5.0978,E2 532.928} C_DIS
LIN {X 15.697,Y -141.5362,Z 180,A -78.8763,B 5.066,C 0.3868,E1 5.1019,E2 531.4511} C_DIS
LIN {X 19.1907,Y -141.1058,Z 180,A -77.4505,B 5.0661,C 0.386,E1 5.1059,E2 530.0232} C_DIS
LIN {X 22.9897,Y -140.5358,Z 180,A -75.9868,B 5.0661,C 0.3862,E1 5.1099,E2 528.5698} C_DIS
LIN {X 26.0767,Y -139.9968,Z 180,A -74.7324,B 5.0661,C 0.3855,E1 5.1133,E2 527.3156} C_DIS
LIN {X 29.4953,Y -139.3161,Z 180,A -73.3319,B 5.0663,C 0.3845,E1 5.1172,E2 525.9144} C_DIS
LIN {X 32.9296,Y -138.5441,Z 180,A -71.94,B 5.0663,C 0.3837,E1 5.121,E2 524.525} C_DIS
LIN {X 36.6407,Y -137.6084,Z 180,A -70.4149,B 5.0663,C 0.3826,E1 5.1251,E2 523.0009} C_DIS
LIN {X 39.988,Y -136.6731,Z 180,A -69.0291,B 5.0665,C 0.3815,E1 5.1288,E2 521.6159} C_DIS
LIN {X 43.0059,Y -135.7541,Z 180,A -67.765,B 5.0665,C 0.3804,E1 5.1322,E2 520.3517} C_DIS
LIN {X 46.6751,Y -134.5363,Z 180,A -66.2309,B 5.0667,C 0.3791,E1 5.1362,E2 518.8194} C_DIS
LIN {X 49.9586,Y -133.3518,Z 180,A -64.8416,B 5.0667,C 0.3777,E1 5.1399,E2 517.4312} C_DIS
LIN {X 52.883,Y -132.2199,Z 180,A -63.5964,B 5.0669,C 0.3765,E1 5.1431,E2 516.1874} C_DIS
LIN {X 56.1326,Y -130.8734,Z 180,A -62.0706,B 5.0671,C 0.3733,E1 5.1471,E2 514.6454} C_DIS
LIN {X 60.2503,Y -129.0299,Z 180,A -60.2887,B 5.0672,C 0.3714,E1 5.1516,E2 512.8668} C_DIS
LIN {X 64.0159,Y -127.2043,Z 180,A -58.6932,B 5.0673,C 0.3703,E1 5.1555,E2 511.2821} C_DIS
LIN {X 67.5789,Y -125.3485,Z 180,A -57.0871,B 5.0675,C 0.3681,E1 5.1595,E2 509.6761} C_DIS
LIN {X 71.1274,Y -123.3697,Z 180,A -55.4229,B 5.0677,C 0.3652,E1 5.1636,E2 508.0066} C_DIS
LIN {X 74.8681,Y -121.1366,Z 180,A -53.6807,B 5.0679,C 0.3626,E1 5.1677,E2 506.2645} C_DIS
LIN {X 78.3898,Y -118.8872,Z 180,A -52.1302,B 5.0679,C 0.3617,E1 5.1713,E2 504.7306} C_DIS
LIN {X 81.4424,Y -116.8172,Z 180,A -50.5785,B 5.0682,C 0.3582,E1 5.1749,E2 503.1684} C_DIS
LIN {X 84.8402,Y -114.3736,Z 180,A -49.0096,B 5.0682,C 0.3568,E1 5.1784,E2 501.6139} C_DIS
LIN {X 88.1632,Y -111.8322,Z 180,A -47.3643,B 5.0684,C 0.3543,E1 5.182,E2 499.9724} C_DIS
LIN {X 91.5462,Y -109.0798,Z 180,A -45.6104,B 5.0687,C 0.351,E1 5.1858,E2 498.2172} C_DIS
LIN {X 94.8604,Y -106.2104,Z 180,A -43.9048,B 5.0689,C 0.3483,E1 5.1894,E2 496.5179} C_DIS
LIN {X 98.0694,Y -103.2555,Z 180,A -42.1424,B 5.0691,C 0.3447,E1 5.193,E2 494.7531} C_DIS
LIN {X 101.1859,Y -100.2027,Z 180,A -40.4466,B 5.0693,C 0.3419,E1 5.1963,E2 493.0639} C_DIS
LIN {X 103.8699,Y -97.4183,Z 180,A -38.8414,B 5.0696,C 0.3379,E1 5.1994,E2 491.4506} C_DIS
LIN {X 106.8052,Y -94.1902,Z 180,A -37.1719,B 5.0697,C 0.3353,E1 5.2025,E2 489.7914} C_DIS
LIN {X 109.6391,Y -90.8756,Z 180,A -35.4292,B 5.07,C 0.3315,E1 5.2056,E2 488.0487} C_DIS
LIN {X 112.3965,Y -87.4426,Z 180,A -33.6905,B 5.0702,C 0.3279,E1 5.2086,E2 486.3129} C_DIS
LIN {X 114.9152,Y -84.1051,Z 180,A -32.039,B 5.0704,C 0.3245,E1 5.2114,E2 484.6642} C_DIS
LIN {X 117.6011,Y -80.3069,Z 180,A -30.229,B 5.0707,C 0.3209,E1 5.2143,E2 482.861} C_DIS
LIN {X 119.9324,Y -76.781,Z 180,A -28.561,B 5.0709,C 0.3172,E1 5.2168,E2 481.1959} C_DIS
LIN {X 122.2231,Y -73.0799,Z 180,A -26.8726,B 5.0711,C 0.3138,E1 5.2192,E2 479.5145} C_DIS
LIN {X 124.42,Y -69.274,Z 180,A -25.1151,B 5.0714,C 0.3095,E1 5.2216,E2 477.7569} C_DIS
LIN {X 126.4926,Y -65.4135,Z 180,A -23.5118,B 5.0715,C 0.3074,E1 5.2237,E2 476.1737} C_DIS
LIN {X 128.0578,Y -62.2926,Z 180,A -21.9954,B 5.0718,C 0.3021,E1 5.2256,E2 474.6409} C_DIS
LIN {X 129.9042,Y -58.3395,Z 180,A -20.3303,B 5.072,C 0.2988,E1 5.2275,E2 472.9864} C_DIS
LIN {X 131.6994,Y -54.1701,Z 180,A -18.6663,B 5.0722,C 0.2964,E1 5.2293,E2 471.343} C_DIS
LIN {X 132.8573,Y -51.2605,Z 180,A -17.4311,B 5.0723,C 0.2934,E1 5.2305,E2 470.1099} C_DIS
LIN {X 134.0731,Y -47.9904,Z 180,A -16.0312,B 5.0725,C 0.2897,E1 5.2319,E2 468.7094} C_DIS
LIN {X 135.472,Y -43.8893,Z 180,A -14.2375,B 5.0729,C 0.2842,E1 5.2335,E2 466.9075} C_DIS
LIN {X 136.8958,Y -39.2275,Z 180,A -12.4662,B 5.0729,C 0.2817,E1 5.2349,E2 465.1601} C_DIS
LIN {X 137.7076,Y -36.2685,Z 180,A -11.2361,B 5.0732,C 0.2783,E1 5.2357,E2 463.9296} C_DIS
LIN {X 138.6351,Y -32.5519,Z 180,A -9.7549,B 5.0734,C 0.2749,E1 5.2367,E2 462.4552} C_DIS
LIN {X 139.3898,Y -29.1496,Z 180,A -8.3783,B 5.0735,C 0.2714,E1 5.2375,E2 461.0809} C_DIS
LIN {X 140.0016,Y -26.0512,Z 180,A -7.1658,B 5.0737,C 0.2687,E1 5.2381,E2 459.8751} C_DIS
LIN {X 140.5985,Y -22.6137,Z 180,A -5.6877,B 5.074,C 0.2636,E1 5.2388,E2 458.3859} C_DIS
LIN {X 141.1558,Y -18.8092,Z 180,A -4.2813,B 5.074,C 0.2614,E1 5.2394,E2 456.9971} C_DIS
LIN {X 141.574,Y -15.3451,Z 180,A -2.9196,B 5.0742,C 0.258,E1 5.2398,E2 455.64} C_DIS
LIN {X 141.9418,Y -11.4663,Z 180,A -1.4367,B 5.0744,C 0.2548,E1 5.2402,E2 454.1673} C_DIS
LIN {X 142.1576,Y -8.3701,Z 180,A -0.2276,B 5.0746,C 0.2519,E1 5.2404,E2 452.9625} C_DIS
LIN {X 142.3268,Y -4.7302,Z 180,A 1.2183,B 5.0747,C 0.248,E1 5.2405,E2 451.5182} C_DIS
LIN {X 142.3985,Y -1.3172,Z 180,A 2.4095,B 5.0747,C 0.2468,E1 5.2405,E2 450.3503} C_DIS
LIN {X 142.3941,Y 1.7418,Z 180,A 3.8004,B 5.0751,C 0.2409,E1 5.2405,E2 448.9371} C_DIS
LIN {X 142.2929,Y 5.6065,Z 180,A 5.2272,B 5.0752,C 0.2384,E1 5.2405,E2 447.5263} C_DIS
LIN {X 142.0883,Y 9.4952,Z 180,A 7.0153,B 5.0756,C 0.2307,E1 5.2401,E2 445.7075} C_DIS
LIN {X 141.7183,Y 13.9545,Z 180,A 8.5802,B 5.0756,C 0.2291,E1 5.2397,E2 444.1728} C_DIS
LIN {X 141.331,Y 17.4515,Z 180,A 9.9306,B 5.0758,C 0.2261,E1 5.2393,E2 442.8302} C_DIS
LIN {X 140.8087,Y 21.2563,Z 180,A 11.4531,B 5.0759,C 0.2221,E1 5.2387,E2 441.3096} C_DIS
LIN {X 140.2454,Y 24.6987,Z 180,A 12.7107,B 5.076,C 0.2203,E1 5.2381,E2 440.0705} C_DIS
LIN {X 139.6061,Y 28.0866,Z 180,A 13.9683,B 5.0761,C 0.2184,E1 5.2375,E2 438.8291} C_DIS
LIN {X 138.8716,Y 31.5173,Z 180,A 15.4506,B 5.0763,C 0.2134,E1 5.2366,E2 437.3367} C_DIS
LIN {X 138.1414,Y 34.5799,Z 180,A 16.8469,B 5.0765,C 0.208,E1 5.2356,E2 435.9223} C_DIS
LIN {X 136.9701,Y 38.9638,Z 180,A 18.6913,B 5.0767,C 0.2027,E1 5.2343,E2 434.0745} C_DIS
LIN {X 135.6448,Y 43.3482,Z 180,A 20.2645,B 5.0767,C 0.2017,E1 5.233,E2 432.5359} C_DIS
LIN {X 134.6577,Y 46.325,Z 180,A 21.6392,B 5.077,C 0.1966,E1 5.2317,E2 431.1455} C_DIS
LIN {X 133.3489,Y 49.9663,Z 180,A 23.0848,B 5.077,C 0.1941,E1 5.2304,E2 429.7138} C_DIS
LIN {X 132.2169,Y 52.8903,Z 180,A 24.3116,B 5.0772,C 0.1913,E1 5.2291,E2 428.4909} C_DIS
LIN {X 130.8825,Y 56.1116,Z 180,A 25.8111,B 5.0774,C 0.1862,E1 5.2275,E2 426.978} C_DIS
LIN {X 129.0293,Y 60.2517,Z 180,A 27.5743,B 5.0775,C 0.1824,E1 5.2254,E2 425.2221} C_DIS
LIN {X 127.2049,Y 64.0148,Z 180,A 29.1498,B 5.0776,C 0.1796,E1 5.2235,E2 423.66} C_DIS
LIN {X 125.5066,Y 67.2847,Z 180,A 30.6306,B 5.0777,C 0.1759,E1 5.2215,E2 422.1787} C_DIS
LIN {X 123.3768,Y 71.115,Z 180,A 32.3847,B 5.0779,C 0.1717,E1 5.2191,E2 420.4251} C_DIS
LIN {X 121.1418,Y 74.8597,Z 180,A 34.1138,B 5.078,C 0.1678,E1 5.2166,E2 418.6988} C_DIS
LIN {X 118.8901,Y 78.3853,Z 180,A 35.6539,B 5.078,C 0.1658,E1 5.2143,E2 417.1768} C_DIS
LIN {X 116.4346,Y 81.9885,Z 180,A 37.3747,B 5.0782,C 0.1622,E1 5.2116,E2 415.4597} C_DIS
LIN {X 113.9655,Y 85.3883,Z 180,A 39.027,B 5.0783,C 0.1588,E1 5.2088,E2 413.812} C_DIS
LIN {X 111.5829,Y 88.4785,Z 180,A 40.6443,B 5.0784,C 0.1546,E1 5.206,E2 412.1879} C_DIS
Enddeposition()
END
